  MoveL 2483 to (5.96, 26.09, 110) mm, rotated rx 180 ry 0 rz 180 deg; joints [-156.697, -51.391, -91.658, 28.324, 56.489, -16.571]
  Call Extruder(23411.01401)
  MoveL 2484 to (0, 26.77, 110) mm, rotated rx 180 ry 0 rz 180 deg; joints [-156.245, -51.047, -92.58, 28.662, 57.126, -16.525]
  Call Extruder(23420.37911)
  MoveL 2485 to (-5.96, 26.09, 110) mm, rotated rx 180 ry 0 rz 180 deg; joints [-155.969, -50.675, -93.588, 28.78, 57.762, -16.332]
  Call Extruder(23429.74391)
  MoveL 2486 to (-11.61, 24.12, 110) mm, rotated rx -180 ry 0 rz 180 deg; joints [-155.891, -50.295, -94.633, 28.669, 58.366, -16.002]
  Call Extruder(23439.10883)
  MoveL 2487 to (-16.69, 20.93, 110) mm, rotated rx 180 ry 0 rz -180 deg; joints [-156.025, -49.925, -95.662, 28.327, 58.909, -15.555]
  Call Extruder(23448.47404)
  MoveL 2488 to (-20.93, 16.69, 110) mm, rotated rx 180 ry 0 rz -180 deg; joints [-156.374, -49.585, -96.624, 27.76, 59.366, -15.014]
  Call Extruder(23457.83895)
  MoveL 2489 to (-24.11, 11.61, 110) mm, rotated rx 180 ry 0 rz 180 deg; joints [-156.928, -49.29, -97.469, 26.989, 59.714, -14.405]
  Call Extruder(23467.20375)
  MoveL 2490 to (-26.09, 5.96, 110) mm, rotated rx 180 ry 0 rz 180 deg; joints [-157.665, -49.055, -98.151, 26.047, 59.935, -13.758]
  Call Extruder(23476.56885)
  MoveL 2491 to (-26.77, 0, 110) mm, rotated rx 180 ry 0 rz 180 deg; joints [-158.546, -48.891, -98.632, 24.978, 60.016, -13.105]
  Call Extruder(23481.35759)
  MoveL 2492 to (-26.42, -3.05, 110) mm, rotated rx -180 ry 0 rz 180 deg; joints [-159.044, -48.846, -98.764, 24.396, 59.984, -12.783]
  Set speed (130.0 mm/s)
  MoveL 2493 to (-41.86, -6.3, 110) mm, rotated rx 180 ry 0 rz -180 deg; joints [-158.606, -47.984, -101.368, 24.484, 61.665, -12.196]
  Call Extruder(23486.35544)
  Set speed (60.0 mm/s)
  MoveL 2494 to (-41.5, -9.47, 110) mm, rotated rx 180 ry 0 rz 180 deg; joints [-159.151, -47.941, -101.503, 23.858, 61.634, -11.866]
  Call Extruder(23501.25108)
  MoveL 2495 to (-38.36, -18.47, 110) mm, rotated rx 180 ry 0 rz 180 deg; joints [-160.835, -47.935, -101.523, 21.976, 61.313, -10.963]
  Call Extruder(23516.14694)
  MoveL 2496 to (-33.29, -26.54, 110) mm, rotated rx -180 ry 0 rz 180 deg; joints [-162.466, -48.056, -101.146, 20.195, 60.776, -10.181]
  Call Extruder(23531.04275)
  MoveL 2497 to (-26.54, -33.28, 110) mm, rotated rx -180 ry 0 rz -180 deg; joints [-163.93, -48.301, -100.397, 18.631, 60.049, -9.555]
  Call Extruder(23545.93861)
  MoveL 2498 to (-18.47, -38.36, 110) mm, rotated rx 180 ry 0 rz 180 deg; joints [-165.137, -48.658, -99.32, 17.381, 59.17, -9.114]
  Call Extruder(23560.83426)
  MoveL 2499 to (-9.47, -41.51, 110) mm, rotated rx -180 ry 0 rz 180 deg; joints [-166.024, -49.114, -97.98, 16.512, 58.184, -8.882]
  Call Extruder(23575.73014)
  MoveL 2500 to (0, -42.57, 110) mm, rotated rx 180 ry 0 rz 180 deg; joints [-166.562, -49.645, -96.451, 16.06, 57.144, -8.877]
  Call Extruder(23586.78613)
  MoveL 2501 to (7.03, -41.78, 110) mm, rotated rx -180 ry 0 rz -180 deg; joints [-166.699, -50.076, -95.239, 16.04, 56.372, -9.047]
  Call Extruder(23590.62601)
  MoveL 2502 to (9.47, -41.51, 110) mm, rotated rx 180 ry 0 rz 180 deg; joints [-166.745, -50.229, -94.815, 16.035, 56.104, -9.106]
  Call Extruder(23605.52167)
  MoveL 2503 to (18.47, -38.36, 110) mm, rotated rx -180 ry 0 rz 180 deg; joints [-166.591, -50.834, -93.155, 16.421, 55.117, -9.567]
  Call Extruder(23620.41752)
  MoveL 2504 to (26.54, -33.29, 110) mm, rotated rx -180 ry 0 rz 180 deg; joints [-166.133, -51.431, -91.553, 17.181, 54.233, -10.244]
  Call Extruder(23635.31333)
  MoveL 2505 to (33.28, -26.54, 110) mm, rotated rx -180 ry 0 rz 180 deg; joints [-165.409, -51.988, -90.083, 18.264, 53.497, -11.107]
  Call Extruder(23650.20919)
  MoveL 2506 to (38.36, -18.47, 110) mm, rotated rx 180 ry 0 rz 180 deg; joints [-164.468, -52.477, -88.814, 19.605, 52.948, -12.112]
  Call Extruder(23665.10484)
  MoveL 2507 to (41.51, -9.47, 110) mm, rotated rx 180 ry 0 rz 180 deg; joints [-163.355, -52.87, -87.803, 21.131, 52.614, -13.207]
  Call Extruder(23680.00071)
  MoveL 2508 to (42.57, 0, 110) mm, rotated rx 180 ry 0 rz 180 deg; joints [-162.12, -53.148, -87.097, 22.765, 52.51, -14.327]
  Call Extruder(23694.89659)
  MoveL 2509 to (41.5, 9.47, 110) mm, rotated rx 180 ry 0 rz 180 deg; joints [-160.81, -53.294, -86.726, 24.427, 52.64, -15.409]
  Call Extruder(23709.79225)
  MoveL 2510 to (38.36, 18.47, 110) mm, rotated rx 180 ry 0 rz 180 deg; joints [-159.475, -53.301, -86.709, 26.043, 52.996, -16.389]
  Call Extruder(23724.68809)
  MoveL 2511 to (33.28, 26.54, 110) mm, rotated rx -180 ry 0 rz -180 deg; joints [-158.16, -53.168, -87.044, 27.544, 53.558, -17.213]
  Call Extruder(23739.58392)
  MoveL 2512 to (26.54, 33.28, 110) mm, rotated rx 180 ry 0 rz 180 deg; joints [-156.916, -52.903, -87.719, 28.872, 54.293, -17.839]
  Call Extruder(23754.47976)
  MoveL 2513 to (18.47, 38.36, 110) mm, rotated rx 180 ry 0 rz -180 deg; joints [-155.789, -52.52, -88.701, 29.976, 55.164, -18.236]
  Call Extruder(23769.37542)
  MoveL 2514 to (9.47, 41.51, 110) mm, rotated rx 180 ry 0 rz 180 deg; joints [-154.828, -52.04, -89.947, 30.816, 56.127, -18.39]
  Call Extruder(23784.27129)
  MoveL 2515 to (0, 42.57, 110) mm, rotated rx 180 ry 0 rz 180 deg; joints [-154.081, -51.489, -91.4, 31.359, 57.134, -18.3]
  Call Extruder(23799.16717)
  MoveL 2516 to (-9.47, 41.51, 110) mm, rotated rx 180 ry 0 rz 180 deg; joints [-153.594, -50.894, -92.992, 31.576, 58.137, -17.976]
  Call Extruder(23814.06282)
  MoveL 2517 to (-18.47, 38.36, 110) mm, rotated rx 180 ry 0 rz -180 deg; joints [-153.408, -50.288, -94.65, 31.448, 59.09, -17.44]
  Call Extruder(23828.95867)
  MoveL 2518 to (-26.54, 33.29, 110) mm, rotated rx 180 ry 0 rz 180 deg; joints [-153.557, -49.701, -96.292, 30.961, 59.949, -16.722]
  Call Extruder(23843.85449)
  MoveL 2519 to (-33.28, 26.54, 110) mm, rotated rx 180 ry 0 rz -180 deg; joints [-154.059, -49.163, -97.835, 30.115, 60.674, -15.859]
  Call Extruder(23858.75034)
  MoveL 2520 to (-38.36, 18.47, 110) mm, rotated rx -180 ry 0 rz 180 deg; joints [-154.913, -48.699, -99.198, 28.928, 61.229, -14.896]
  Call Extruder(23873.64600)
  MoveL 2521 to (-41.5, 9.47, 110) mm, rotated rx 180 ry 0 rz 180 deg; joints [-156.091, -48.331, -100.303, 27.439, 61.587, -13.877]
  Call Extruder(23888.54187)
  MoveL 2522 to (-42.57, 0, 110) mm, rotated rx 180 ry 0 rz -180 deg; joints [-157.533, -48.075, -101.088, 25.717, 61.726, -12.852]
  Call Extruder(23896.09615)
  MoveL 2523 to (-42.03, -4.8, 110) mm, rotated rx -180 ry 0 rz 180 deg; joints [-158.35, -48.005, -101.304, 24.777, 61.679, -12.351]
  Set speed (130.0 mm/s)
  MoveL 2524 to (-54.1, -7.67, 110) mm, rotated rx -180 ry 0 rz 180 deg; joints [-158.024, -47.368, -103.323, 24.834, 63.002, -11.865]
  Call Extruder(23900.16878)
  Set speed (30.0 mm/s)
  MoveL 2525 to (-53.59, -12.23, 110) mm, rotated rx 180 ry 0 rz 180 deg; joints [-158.835, -47.307, -103.518, 23.914, 62.961, -11.397]
  Call Extruder(23911.09891)
  MoveL 2526 to (-49.52, -23.85, 110) mm, rotated rx 180 ry 0 rz 180 deg; joints [-161.095, -47.299, -103.544, 21.413, 62.554, -10.246]
  Call Extruder(23922.02920)
  MoveL 2527 to (-42.98, -34.27, 110) mm, rotated rx 180 ry 0 rz 180 deg; joints [-163.275, -47.453, -103.047, 19.047, 61.862, -9.248]
  Call Extruder(23932.95931)
  MoveL 2528 to (-34.27, -42.98, 110) mm, rotated rx -180 ry 0 rz 180 deg; joints [-165.21, -47.763, -102.059, 16.983, 60.92, -8.443]
  Call Extruder(23943.88960)
  MoveL 2529 to (-23.85, -49.52, 110) mm, rotated rx 180 ry 0 rz 180 deg; joints [-166.774, -48.219, -100.647, 15.354, 59.779, -7.869]
  Call Extruder(23954.81973)
  MoveL 2530 to (-12.23, -53.59, 110) mm, rotated rx -180 ry 0 rz 180 deg; joints [-167.889, -48.801, -98.897, 14.245, 58.5, -7.556]
  Call Extruder(23965.74996)
  MoveL 2531 to (0, -54.97, 110) mm, rotated rx 180 ry 0 rz 180 deg; joints [-168.526, -49.485, -96.91, 13.696, 57.152, -7.53]
  Call Extruder(23973.26563)
  MoveL 2532 to (8.41, -54.02, 110) mm, rotated rx -180 ry 0 rz -180 deg; joints [-168.645, -49.998, -95.458, 13.702, 56.225, -7.719]
  Call Extruder(23976.68018)
  MoveL 2533 to (12.23, -53.59, 110) mm, rotated rx -180 ry 0 rz 180 deg; joints [-168.697, -50.237, -94.793, 13.708, 55.804, -7.806]
  Call Extruder(23987.61032)
  MoveL 2534 to (23.85, -49.53, 110) mm, rotated rx 180 ry 0 rz 180 deg; joints [-168.436, -51.019, -92.655, 14.25, 54.524, -8.384]
  Call Extruder(23998.54060)
  MoveL 2535 to (34.27, -42.98, 110) mm, rotated rx 180 ry 0 rz 180 deg; joints [-167.797, -51.793, -90.596, 15.27, 53.379, -9.249]
  Call Extruder(24009.47072)
  MoveL 2536 to (42.98, -34.27, 110) mm, rotated rx 180 ry 0 rz 180 deg; joints [-166.837, -52.516, -88.711, 16.697, 52.427, -10.365]
  Call Extruder(24020.40100)
  MoveL 2537 to (49.53, -23.85, 110) mm, rotated rx -180 ry 0 rz 180 deg; joints [-165.618, -53.151, -87.087, 18.447, 51.717, -11.676]
  Call Extruder(24031.33113)
  MoveL 2538 to (53.59, -12.23, 110) mm, rotated rx -180 ry 0 rz -180 deg; joints [-164.2, -53.663, -85.795, 20.423, 51.285, -13.11]
  Call Extruder(24042.26136)
  MoveL 2539 to (54.97, 0, 110) mm, rotated rx -180 ry 0 rz 180 deg; joints [-162.641, -54.025, -84.892, 22.525, 51.154, -14.581]
  Call Extruder(24053.19158)
  MoveL 2540 to (53.59, 12.23, 110) mm, rotated rx 180 ry 0 rz 180 deg; joints [-160.996, -54.215, -84.418, 24.65, 51.329, -16]
  Call Extruder(24064.12172)
  MoveL 2541 to (49.52, 23.85, 110) mm, rotated rx 180 ry 0 rz -180 deg; joints [-159.322, -54.224, -84.396, 26.703, 51.796, -17.28]
  Call Extruder(24075.05200)
  MoveL 2542 to (42.98, 34.27, 110) mm, rotated rx 180 ry 0 rz 180 deg; joints [-157.673, -54.052, -84.825, 28.599, 52.528, -18.35]
  Call Extruder(24085.98212)
  MoveL 2543 to (34.27, 42.98, 110) mm, rotated rx 180 ry 0 rz 180 deg; joints [-156.102, -53.706, -85.687, 30.269, 53.483, -19.152]
  Call Extruder(24096.91240)
  MoveL 2544 to (23.85, 49.52, 110) mm, rotated rx -180 ry 0 rz 180 deg; joints [-154.667, -53.208, -86.943, 31.658, 54.609, -19.652]
  Call Extruder(24107.84254)
  MoveL 2545 to (12.23, 53.59, 110) mm, rotated rx -180 ry 0 rz 180 deg; joints [-153.426, -52.584, -88.537, 32.722, 55.85, -19.834]
  Call Extruder(24118.77276)
  MoveL 2546 to (0, 54.97, 110) mm, rotated rx 180 ry 0 rz 180 deg; joints [-152.438, -51.868, -90.399, 33.423, 57.144, -19.7]
  Call Extruder(24129.70298)
  MoveL 2547 to (-12.23, 53.59, 110) mm, rotated rx 180 ry 0 rz 180 deg; joints [-151.764, -51.097, -92.445, 33.73, 58.431, -19.267]
  Call Extruder(24140.63312)
  MoveL 2548 to (-23.85, 49.52, 110) mm, rotated rx 180 ry 0 rz 180 deg; joints [-151.463, -50.313, -94.58, 33.612, 59.654, -18.563]
  Call Extruder(24151.56340)
  MoveL 2549 to (-34.27, 42.98, 110) mm, rotated rx 180 ry 0 rz 180 deg; joints [-151.589, -49.557, -96.704, 33.044, 60.756, -17.63]
  Call Extruder(24162.49352)
  MoveL 2550 to (-42.98, 34.27, 110) mm, rotated rx 180 ry 0 rz -180 deg; joints [-152.179, -48.865, -98.708, 32.013, 61.69, -16.514]
  Call Extruder(24173.42380)
  MoveL 2551 to (-49.53, 23.85, 110) mm, rotated rx -180 ry 0 rz -180 deg; joints [-153.248, -48.271, -100.487, 30.523, 62.41, -15.273]
  Call Extruder(24184.35394)
  MoveL 2552 to (-53.59, 12.23, 110) mm, rotated rx -180 ry 0 rz -180 deg; joints [-154.769, -47.802, -101.937, 28.615, 62.879, -13.966]
  Call Extruder(24195.28416)
  MoveL 2553 to (-54.97, 0, 110) mm, rotated rx 180 ry 0 rz -180 deg; joints [-156.673, -47.477, -102.97, 26.369, 63.069, -12.655]
  Call Extruder(24200.80978)
  MoveL 2554 to (-54.27, -6.18, 110) mm, rotated rx 180 ry 0 rz 180 deg; joints [-157.76, -47.388, -103.256, 25.134, 63.015, -12.018]
  Set speed (130.0 mm/s)
  MoveL 2555 to (-49.9, -9.51, 110) mm, rotated rx -180 ry 0 rz 180 deg; joints [-158.616, -47.532, -102.794, 24.26, 62.549, -11.736]
  MoveL 2556 to (2.97, -12.99, 110) mm, rotated rx -180 ry 0 rz -180 deg; joints [-162.152, -50.315, -94.576, 21.484, 56.807, -12.16]
  Call Extruder(24205.47337)
  Set speed (80.0 mm/s)
  MoveL 2557 to (5.78, -12.01, 110) mm, rotated rx -180 ry 0 rz 180 deg; joints [-162.141, -50.504, -94.055, 21.578, 56.501, -12.313]
  Call Extruder(24210.13699)
  MoveL 2558 to (8.31, -10.42, 110) mm, rotated rx -180 ry 0 rz -180 deg; joints [-162.027, -50.69, -93.547, 21.791, 56.227, -12.53]
  Call Extruder(24214.80118)
  MoveL 2559 to (10.42, -8.31, 110) mm, rotated rx 180 ry 0 rz 180 deg; joints [-161.819, -50.862, -93.079, 22.109, 55.998, -12.799]
  Call Extruder(24219.46481)
  MoveL 2560 to (12.01, -5.78, 110) mm, rotated rx -180 ry 0 rz 180 deg; joints [-161.529, -51.013, -92.673, 22.517, 55.826, -13.108]
  Call Extruder(24224.12838)
  MoveL 2561 to (13, -2.97, 110) mm, rotated rx -180 ry 0 rz -180 deg; joints [-161.171, -51.133, -92.348, 22.992, 55.72, -13.441]
  Call Extruder(24228.79233)
  MoveL 2562 to (13.33, 0, 110) mm, rotated rx -180 ry 0 rz 180 deg; joints [-160.763, -51.218, -92.12, 23.51, 55.685, -13.779]
  Call Extruder(24233.45628)
  MoveL 2563 to (12.99, 2.97, 110) mm, rotated rx -180 ry 0 rz 180 deg; joints [-160.324, -51.263, -92, 24.046, 55.722, -14.107]
  Call Extruder(24238.11985)
  MoveL 2564 to (12.01, 5.78, 110) mm, rotated rx 180 ry 0 rz -180 deg; joints [-159.874, -51.265, -91.995, 24.575, 55.83, -14.405]
  Call Extruder(24242.78348)
  MoveL 2565 to (10.42, 8.31, 110) mm, rotated rx 180 ry 0 rz 180 deg; joints [-159.432, -51.225, -92.103, 25.071, 56.002, -14.66]
  Call Extruder(24247.44767)
  MoveL 2566 to (8.31, 10.42, 110) mm, rotated rx 180 ry 0 rz -180 deg; joints [-159.021, -51.144, -92.321, 25.512, 56.23, -14.857]
  Call Extruder(24252.11129)
  MoveL 2567 to (5.78, 12.01, 110) mm, rotated rx 180 ry 0 rz 180 deg; joints [-158.657, -51.026, -92.637, 25.877, 56.502, -14.987]
  Call Extruder(24256.77487)
  MoveL 2568 to (2.97, 13, 110) mm, rotated rx 180 ry 0 rz -180 deg; joints [-158.359, -50.878, -93.036, 26.149, 56.805, -15.045]
  Call Extruder(24261.43882)
  MoveL 2569 to (0, 13.33, 110) mm, rotated rx -180 ry 0 rz -180 deg; joints [-158.143, -50.708, -93.499, 26.314, 57.124, -15.026]
  Call Extruder(24266.10278)
  MoveL 2570 to (-2.97, 13, 110) mm, rotated rx 180 ry 0 rz 180 deg; joints [-158.019, -50.523, -94.003, 26.365, 57.443, -14.934]
  Call Extruder(24270.76634)
  MoveL 2571 to (-5.78, 12.01, 110) mm, rotated rx 180 ry 0 rz 180 deg; joints [-157.997, -50.334, -94.524, 26.296, 57.745, -14.774]
  Call Extruder(24275.42997)
  MoveL 2572 to (-8.31, 10.42, 110) mm, rotated rx -180 ry 0 rz 180 deg; joints [-158.08, -50.149, -95.035, 26.111, 58.018, -14.553]
  Call Extruder(24280.09417)
  MoveL 2573 to (-10.42, 8.31, 110) mm, rotated rx 180 ry 0 rz 180 deg; joints [-158.266, -49.979, -95.511, 25.816, 58.246, -14.284]
  Call Extruder(24284.75779)
  MoveL 2574 to (-12.01, 5.78, 110) mm, rotated rx 180 ry 0 rz 180 deg; joints [-158.549, -49.831, -95.927, 25.423, 58.418, -13.979]
  Call Extruder(24289.42136)
  MoveL 2575 to (-13, 2.97, 110) mm, rotated rx 180 ry 0 rz -180 deg; joints [-158.913, -49.713, -96.261, 24.951, 58.526, -13.654]
  Call Extruder(24294.08531)
  MoveL 2576 to (-13.33, 0, 110) mm, rotated rx 180 ry 0 rz 180 deg; joints [-159.341, -49.63, -96.496, 24.424, 58.565, -13.324]
  Call Extruder(24298.74927)
  MoveL 2577 to (-12.99, -2.97, 110) mm, rotated rx -180 ry 0 rz 180 deg; joints [-159.811, -49.586, -96.62, 23.868, 58.531, -13.006]
  Call Extruder(24303.41283)
  MoveL 2578 to (-12.01, -5.78, 110) mm, rotated rx 180 ry 0 rz 180 deg; joints [-160.294, -49.584, -96.626, 23.314, 58.427, -12.715]
  Call Extruder(24308.07647)
  MoveL 2579 to (-10.42, -8.31, 110) mm, rotated rx 180 ry 0 rz 180 deg; joints [-160.766, -49.623, -96.514, 22.791, 58.257, -12.465]
  Call Extruder(24312.74065)
  MoveL 2580 to (-8.31, -10.42, 110) mm, rotated rx 180 ry 0 rz 180 deg; joints [-161.2, -49.703, -96.289, 22.327, 58.03, -12.268]
  Call Extruder(24317.40429)
  MoveL 2581 to (-5.78, -12.01, 110) mm, rotated rx 180 ry 0 rz 180 deg; joints [-161.572, -49.818, -95.964, 21.947, 57.757, -12.133]
  Call Extruder(24322.06785)
  MoveL 2582 to (-2.97, -13, 110) mm, rotated rx 180 ry 0 rz 180 deg; joints [-161.863, -49.963, -95.555, 21.673, 57.452, -12.068]
  Call Extruder(24326.73181)
  MoveL 2583 to (0, -13.33, 110) mm, rotated rx 180 ry 0 rz -180 deg; joints [-162.059, -50.132, -95.084, 21.516, 57.13, -12.077]
  Call Extruder(24331.39575)
  MoveL 2584 to (2.97, -12.99, 110) mm, rotated rx -180 ry 0 rz -180 deg; joints [-162.152, -50.315, -94.576, 21.484, 56.807, -12.16]
  Set speed (130.0 mm/s)
  MoveL 2585 to (2.97, -12.99, 115) mm, rotated rx 180 ry 0 rz -180 deg; joints [-162.152, -49.558, -94.868, 21.597, 56.374, -12.365]
  MoveL 2586 to (-26.25, -4.54, 115) mm, rotated rx 180 ry 0 rz 180 deg; joints [-159.288, -48.032, -99.127, 24.229, 59.519, -12.859]
  Call Extruder(24333.62836)
  Set speed (60.0 mm/s)
  MoveL 2587 to (-26.09, -5.96, 115) mm, rotated rx 180 ry 0 rz 180 deg; joints [-159.522, -48.012, -99.186, 23.955, 59.502, -12.707]
  Call Extruder(24342.99315)
  MoveL 2588 to (-24.11, -11.61, 115) mm, rotated rx 180 ry 0 rz 180 deg; joints [-160.532, -48.007, -99.199, 22.808, 59.293, -12.12]
  Call Extruder(24352.35808)
  MoveL 2589 to (-20.93, -16.69, 115) mm, rotated rx -180 ry 0 rz 180 deg; joints [-161.513, -48.087, -98.968, 21.723, 58.951, -11.612]
  Call Extruder(24361.72328)
  MoveL 2590 to (-16.69, -20.93, 115) mm, rotated rx 180 ry 0 rz 180 deg; joints [-162.406, -48.248, -98.507, 20.764, 58.495, -11.207]
  Call Extruder(24371.08820)
  MoveL 2591 to (-11.61, -24.12, 115) mm, rotated rx 180 ry 0 rz 180 deg; joints [-163.159, -48.482, -97.842, 19.988, 57.946, -10.926]
  Call Extruder(24380.45299)
  MoveL 2592 to (-5.96, -26.09, 115) mm, rotated rx -180 ry 0 rz 180 deg; joints [-163.733, -48.779, -97.01, 19.435, 57.334, -10.783]
  Call Extruder(24389.81809)
  MoveL 2593 to (0, -26.77, 115) mm, rotated rx 180 ry 0 rz 180 deg; joints [-164.103, -49.123, -96.056, 19.133, 56.689, -10.787]
  Call Extruder(24399.18321)
  MoveL 2594 to (5.96, -26.09, 115) mm, rotated rx -180 ry 0 rz 180 deg; joints [-164.258, -49.498, -95.029, 19.092, 56.044, -10.942]
  Call Extruder(24408.54800)
  MoveL 2595 to (11.61, -24.11, 115) mm, rotated rx -180 ry 0 rz 180 deg; joints [-164.201, -49.886, -93.982, 19.307, 55.433, -11.242]
  Call Extruder(24417.91291)
  MoveL 2596 to (16.69, -20.93, 115) mm, rotated rx 180 ry 0 rz 180 deg; joints [-163.944, -50.267, -92.967, 19.762, 54.886, -11.676]
  Call Extruder(24427.27812)
  MoveL 2597 to (20.93, -16.69, 115) mm, rotated rx 180 ry 0 rz 180 deg; joints [-163.508, -50.622, -92.033, 20.426, 54.433, -12.222]
  Call Extruder(24436.64304)
  MoveL 2598 to (24.12, -11.61, 115) mm, rotated rx 180 ry 0 rz 180 deg; joints [-162.92, -50.932, -91.224, 21.261, 54.094, -12.854]
  Call Extruder(24446.00784)
  MoveL 2599 to (26.09, -5.96, 115) mm, rotated rx -180 ry 0 rz -180 deg; joints [-162.209, -51.181, -90.579, 22.222, 53.889, -13.538]
  Call Extruder(24455.37293)
  MoveL 2600 to (26.77, 0, 115) mm, rotated rx -180 ry 0 rz -180 deg; joints [-161.41, -51.356, -90.128, 23.261, 53.826, -14.237]
  Call Extruder(24464.73804)
  MoveL 2601 to (26.09, 5.96, 115) mm, rotated rx -180 ry 0 rz -180 deg; joints [-160.556, -51.449, -89.891, 24.327, 53.909, -14.912]
  Call Extruder(24474.10285)
  MoveL 2602 to (24.11, 11.61, 115) mm, rotated rx -180 ry 0 rz 180 deg; joints [-159.683, -51.453, -89.88, 25.37, 54.132, -15.528]
  Call Extruder(24483.46775)
  MoveL 2603 to (20.93, 16.69, 115) mm, rotated rx 180 ry 0 rz 180 deg; joints [-158.826, -51.369, -90.095, 26.345, 54.483, -16.05]
  Call Extruder(24492.83297)
  MoveL 2604 to (16.69, 20.93, 115) mm, rotated rx 180 ry 0 rz 180 deg; joints [-158.019, -51.202, -90.525, 27.209, 54.944, -16.452]
  Call Extruder(24502.19787)
  MoveL 2605 to (11.61, 24.12, 115) mm, rotated rx -180 ry 0 rz 180 deg; joints [-157.299, -50.96, -91.152, 27.926, 55.49, -16.715]
  Call Extruder(24511.56268)
  MoveL 2606 to (5.96, 26.09, 115) mm, rotated rx -180 ry 0 rz 180 deg; joints [-156.697, -50.655, -91.946, 28.466, 56.095, -16.827]
  Call Extruder(24520.92778)
  MoveL 2607 to (0, 26.77, 115) mm, rotated rx 180 ry 0 rz -180 deg; joints [-156.245, -50.304, -92.87, 28.804, 56.728, -16.786]
  Call Extruder(24530.29289)
  MoveL 2608 to (-5.96, 26.09, 115) mm, rotated rx 180 ry 0 rz 180 deg; joints [-155.969, -49.925, -93.879, 28.921, 57.359, -16.594]
  Call Extruder(24539.65768)
  MoveL 2609 to (-11.61, 24.12, 115) mm, rotated rx 180 ry 0 rz -180 deg; joints [-155.891, -49.537, -94.925, 28.809, 57.958, -16.266]
  Call Extruder(24549.02260)
  MoveL 2610 to (-16.69, 20.93, 115) mm, rotated rx 180 ry 0 rz -180 deg; joints [-156.025, -49.159, -95.956, 28.463, 58.494, -15.818]
  Call Extruder(24558.38781)
  MoveL 2611 to (-20.93, 16.69, 115) mm, rotated rx 180 ry 0 rz 180 deg; joints [-156.374, -48.811, -96.92, 27.894, 58.944, -15.273]
  Call Extruder(24567.75272)
  MoveL 2612 to (-24.11, 11.61, 115) mm, rotated rx -180 ry 0 rz 180 deg; joints [-156.928, -48.509, -97.766, 27.119, 59.283, -14.66]
  Call Extruder(24577.11752)
  MoveL 2613 to (-26.09, 5.96, 115) mm, rotated rx 180 ry 0 rz -180 deg; joints [-157.665, -48.268, -98.449, 26.172, 59.496, -14.007]
  Call Extruder(24586.48263)
  MoveL 2614 to (-26.77, 0, 115) mm, rotated rx 180 ry 0 rz -180 deg; joints [-158.546, -48.1, -98.932, 25.099, 59.571, -13.346]
  Call Extruder(24591.27137)
  MoveL 2615 to (-26.42, -3.05, 115) mm, rotated rx 180 ry 0 rz 180 deg; joints [-159.044, -48.054, -99.064, 24.515, 59.536, -13.019]
  Set speed (130.0 mm/s)
  MoveL 2616 to (-41.86, -6.3, 115) mm, rotated rx -180 ry 0 rz 180 deg; joints [-158.606, -47.168, -101.674, 24.6, 61.201, -12.438]
  Call Extruder(24596.26921)
  Set speed (60.0 mm/s)
  MoveL 2617 to (-41.51, -9.47, 115) mm, rotated rx 180 ry 0 rz -180 deg; joints [-159.151, -47.124, -101.809, 23.97, 61.167, -12.102]
  Call Extruder(24611.16485)
  MoveL 2618 to (-38.36, -18.47, 115) mm, rotated rx 180 ry 0 rz 180 deg; joints [-160.835, -47.117, -101.829, 22.082, 60.839, -11.182]
  Call Extruder(24626.06071)
  MoveL 2619 to (-33.28, -26.54, 115) mm, rotated rx 180 ry 0 rz 180 deg; joints [-162.466, -47.242, -101.451, 20.294, 60.299, -10.383]
  Call Extruder(24640.95653)
  MoveL 2620 to (-26.54, -33.28, 115) mm, rotated rx -180 ry 0 rz -180 deg; joints [-163.93, -47.494, -100.7, 18.725, 59.572, -9.741]
  Call Extruder(24655.85238)
  MoveL 2621 to (-18.47, -38.36, 115) mm, rotated rx -180 ry 0 rz 180 deg; joints [-165.137, -47.862, -99.621, 17.471, 58.697, -9.287]
  Call Extruder(24670.74803)
  MoveL 2622 to (-9.47, -41.5, 115) mm, rotated rx 180 ry 0 rz 180 deg; joints [-166.024, -48.328, -98.278, 16.599, 57.718, -9.046]
  Call Extruder(24685.64390)
  MoveL 2623 to (0, -42.57, 115) mm, rotated rx 180 ry 0 rz 180 deg; joints [-166.562, -48.873, -96.746, 16.146, 56.686, -9.035]
  Call Extruder(24697.35594)
  MoveL 2624 to (7.45, -41.73, 115) mm, rotated rx 180 ry 0 rz 180 deg; joints [-166.707, -49.34, -95.46, 16.126, 55.876, -9.213]
  Call Extruder(24700.53978)
  MoveL 2625 to (9.47, -41.51, 115) mm, rotated rx 180 ry 0 rz 180 deg; joints [-166.745, -49.469, -95.108, 16.123, 55.656, -9.262]
  Call Extruder(24715.43544)
  MoveL 2626 to (18.47, -38.36, 115) mm, rotated rx -180 ry 0 rz 180 deg; joints [-166.591, -50.087, -93.445, 16.512, 54.678, -9.725]
  Call Extruder(24730.33128)
  MoveL 2627 to (26.54, -33.28, 115) mm, rotated rx 180 ry 0 rz 180 deg; joints [-166.133, -50.695, -91.84, 17.277, 53.805, -10.408]
  Call Extruder(24745.22710)
  MoveL 2628 to (33.29, -26.54, 115) mm, rotated rx 180 ry 0 rz -180 deg; joints [-165.409, -51.263, -90.369, 18.367, 53.08, -11.279]
  Call Extruder(24760.12296)
  MoveL 2629 to (38.36, -18.47, 115) mm, rotated rx 180 ry 0 rz 180 deg; joints [-164.468, -51.759, -89.098, 19.715, 52.541, -12.295]
  Call Extruder(24775.01861)
  MoveL 2630 to (41.5, -9.47, 115) mm, rotated rx -180 ry 0 rz 180 deg; joints [-163.355, -52.159, -88.087, 21.25, 52.215, -13.402]
  Call Extruder(24789.91448)
  MoveL 2631 to (42.57, 0, 115) mm, rotated rx 180 ry 0 rz 180 deg; joints [-162.12, -52.441, -87.38, 22.892, 52.119, -14.535]
  Call Extruder(24804.81036)
  MoveL 2632 to (41.51, 9.47, 115) mm, rotated rx 180 ry 0 rz 180 deg; joints [-160.81, -52.589, -87.009, 24.562, 52.256, -15.629]
  Call Extruder(24819.70602)
  MoveL 2633 to (38.36, 18.47, 115) mm, rotated rx 180 ry 0 rz 180 deg; joints [-159.475, -52.596, -86.991, 26.184, 52.618, -16.622]
  Call Extruder(24834.60186)
  MoveL 2634 to (33.29, 26.54, 115) mm, rotated rx -180 ry 0 rz -180 deg; joints [-158.16, -52.462, -87.328, 27.69, 53.183, -17.458]
  Call Extruder(24849.49768)
  MoveL 2635 to (26.54, 33.28, 115) mm, rotated rx 180 ry 0 rz 180 deg; joints [-156.916, -52.193, -88.002, 29.021, 53.92, -18.094]
  Call Extruder(24864.39353)
  MoveL 2636 to (18.47, 38.36, 115) mm, rotated rx 180 ry 0 rz -180 deg; joints [-155.789, -51.804, -88.985, 30.128, 54.79, -18.5]
  Call Extruder(24879.28919)
  MoveL 2637 to (9.47, 41.5, 115) mm, rotated rx 180 ry 0 rz 180 deg; joints [-154.828, -51.316, -90.233, 30.968, 55.75, -18.662]
  Call Extruder(24894.18507)
  MoveL 2638 to (0, 42.57, 115) mm, rotated rx 180 ry 0 rz 180 deg; joints [-154.081, -50.754, -91.687, 31.51, 56.752, -18.578]
  Call Extruder(24909.08094)
  MoveL 2639 to (-9.47, 41.51, 115) mm, rotated rx 180 ry 0 rz 180 deg; joints [-153.594, -50.148, -93.282, 31.726, 57.749, -18.258]
  Call Extruder(24923.97659)
  MoveL 2640 to (-18.47, 38.36, 115) mm, rotated rx -180 ry 0 rz -180 deg; joints [-153.408, -49.53, -94.943, 31.595, 58.693, -17.725]
  Call Extruder(24938.87244)
  MoveL 2641 to (-26.54, 33.29, 115) mm, rotated rx 180 ry 0 rz 180 deg; joints [-153.557, -48.93, -96.587, 31.104, 59.541, -17.006]
  Call Extruder(24953.76826)
  MoveL 2642 to (-33.28, 26.54, 115) mm, rotated rx 180 ry 0 rz 180 deg; joints [-154.059, -48.379, -98.133, 30.254, 60.254, -16.14]
  Call Extruder(24968.66411)
  MoveL 2643 to (-38.36, 18.47, 115) mm, rotated rx -180 ry 0 rz -180 deg; joints [-154.913, -47.904, -99.499, 29.061, 60.796, -15.17]
  Call Extruder(24983.55977)
  MoveL 2644 to (-41.5, 9.47, 115) mm, rotated rx 180 ry 0 rz -180 deg; joints [-156.091, -47.526, -100.607, 27.565, 61.141, -14.142]
  Call Extruder(24998.45564)
  MoveL 2645 to (-42.57, 0, 115) mm, rotated rx 180 ry 0 rz -180 deg; joints [-157.533, -47.262, -101.393, 25.837, 61.268, -13.103]
  Call Extruder(25006.00993)
  MoveL 2646 to (-42.03, -4.8, 115) mm, rotated rx -180 ry 0 rz 180 deg; joints [-158.35, -47.19, -101.609, 24.894, 61.217, -12.595]
  Set speed (130.0 mm/s)
  MoveL 2647 to (-54.1, -7.67, 115) mm, rotated rx 180 ry 0 rz -180 deg; joints [-158.024, -46.533, -103.633, 24.948, 62.526, -12.113]
  Call Extruder(25010.08255)
  Set speed (30.0 mm/s)
  MoveL 2648 to (-53.59, -12.23, 115) mm, rotated rx 180 ry 0 rz -180 deg; joints [-158.835, -46.47, -103.829, 24.024, 62.481, -11.637]
  Call Extruder(25021.01269)
  MoveL 2649 to (-49.53, -23.85, 115) mm, rotated rx -180 ry 0 rz 180 deg; joints [-161.095, -46.462, -103.855, 21.514, 62.064, -10.463]
  Call Extruder(25031.94297)
  MoveL 2650 to (-42.98, -34.27, 115) mm, rotated rx 180 ry 0 rz 180 deg; joints [-163.275, -46.621, -103.356, 19.14, 61.368, -9.442]
  Call Extruder(25042.87309)
  MoveL 2651 to (-34.27, -42.98, 115) mm, rotated rx -180 ry 0 rz 180 deg; joints [-165.21, -46.941, -102.367, 17.068, 60.428, -8.616]
  Call Extruder(25053.80337)
  MoveL 2652 to (-23.85, -49.53, 115) mm, rotated rx -180 ry 0 rz 180 deg; joints [-166.774, -47.41, -100.951, 15.433, 59.292, -8.024]
  Call Extruder(25064.73351)
  MoveL 2653 to (-12.23, -53.59, 115) mm, rotated rx 180 ry 0 rz 180 deg; joints [-167.889, -48.008, -99.197, 14.32, 58.023, -7.699]
  Call Extruder(25075.66373)
  MoveL 2654 to (0, -54.97, 115) mm, rotated rx -180 ry 0 rz 180 deg; joints [-168.526, -48.708, -97.206, 13.77, 56.686, -7.666]
  Call Extruder(25083.55224)
  MoveL 2655 to (8.83, -53.97, 115) mm, rotated rx -180 ry 0 rz -180 deg; joints [-168.651, -49.26, -95.679, 13.778, 55.722, -7.863]
  Call Extruder(25086.59395)
  MoveL 2656 to (12.23, -53.59, 115) mm, rotated rx -180 ry 0 rz 180 deg; joints [-168.697, -49.477, -95.086, 13.784, 55.35, -7.94]
  Call Extruder(25097.52409)
  MoveL 2657 to (23.85, -49.53, 115) mm, rotated rx -180 ry 0 rz 180 deg; joints [-168.436, -50.276, -92.944, 14.33, 54.084, -8.522]
  Call Extruder(25108.45437)
  MoveL 2658 to (34.27, -42.98, 115) mm, rotated rx -180 ry 0 rz 180 deg; joints [-167.797, -51.064, -90.882, 15.357, 52.953, -9.395]
  Call Extruder(25119.38449)
  MoveL 2659 to (42.98, -34.27, 115) mm, rotated rx -180 ry 0 rz 180 deg; joints [-166.837, -51.8, -88.996, 16.794, 52.013, -10.523]
  Call Extruder(25130.31477)
  MoveL 2660 to (49.53, -23.85, 115) mm, rotated rx -180 ry 0 rz 180 deg; joints [-165.618, -52.445, -87.37, 18.554, 51.315, -11.848]
  Call Extruder(25141.24491)
  MoveL 2661 to (53.59, -12.23, 115) mm, rotated rx 180 ry 0 rz -180 deg; joints [-164.2, -52.964, -86.077, 20.541, 50.894, -13.298]
  Call Extruder(25152.17513)
  MoveL 2662 to (54.97, 0, 115) mm, rotated rx 180 ry 0 rz 180 deg; joints [-162.641, -53.331, -85.173, 22.654, 50.773, -14.785]
  Call Extruder(25163.10535)
  MoveL 2663 to (53.59, 12.23, 115) mm, rotated rx 180 ry 0 rz 180 deg; joints [-160.996, -53.524, -84.7, 24.788, 50.956, -16.22]
  Call Extruder(25174.03549)
  MoveL 2664 to (49.52, 23.85, 115) mm, rotated rx -180 ry 0 rz -180 deg; joints [-159.322, -53.533, -84.677, 26.849, 51.43, -17.516]
  Call Extruder(25184.96577)
  MoveL 2665 to (42.98, 34.27, 115) mm, rotated rx 180 ry 0 rz 180 deg; joints [-157.673, -53.358, -85.107, 28.751, 52.166, -18.599]
  Call Extruder(25195.89589)
  MoveL 2666 to (34.27, 42.98, 115) mm, rotated rx -180 ry 0 rz -180 deg; joints [-156.102, -53.008, -85.969, 30.426, 53.123, -19.415]
  Call Extruder(25206.82617)
  MoveL 2667 to (23.85, 49.53, 115) mm, rotated rx 180 ry 0 rz -180 deg; joints [-154.667, -52.502, -87.226, 31.818, 54.25, -19.926]
  Call Extruder(25217.75631)
  MoveL 2668 to (12.23, 53.59, 115) mm, rotated rx -180 ry 0 rz 180 deg; joints [-153.426, -51.868, -88.822, 32.882, 55.487, -20.117]
  Call Extruder(25228.68653)
  MoveL 2669 to (0, 54.97, 115) mm, rotated rx 180 ry 0 rz 180 deg; joints [-152.438, -51.14, -90.686, 33.582, 56.776, -19.99]
  Call Extruder(25239.61676)
  MoveL 2670 to (-12.23, 53.59, 115) mm, rotated rx -180 ry 0 rz 180 deg; joints [-151.764, -50.355, -92.734, 33.886, 58.055, -19.563]
  Call Extruder(25250.54689)
  MoveL 2671 to (-23.85, 49.52, 115) mm, rotated rx -180 ry 0 rz 180 deg; joints [-151.463, -49.556, -94.873, 33.764, 59.266, -18.863]
  Call Extruder(25261.47717)
  MoveL 2672 to (-34.27, 42.98, 115) mm, rotated rx 180 ry 0 rz 180 deg; joints [-151.589, -48.782, -96.999, 33.192, 60.356, -17.93]
  Call Extruder(25272.40729)
  MoveL 2673 to (-42.98, 34.27, 115) mm, rotated rx -180 ry 0 rz -180 deg; joints [-152.179, -48.073, -99.008, 32.155, 61.273, -16.812]
  Call Extruder(25283.33757)
  MoveL 2674 to (-49.52, 23.85, 115) mm, rotated rx 180 ry 0 rz 180 deg; joints [-153.248, -47.464, -100.79, 30.659, 61.976, -15.563]
  Call Extruder(25294.26771)
  MoveL 2675 to (-53.59, 12.23, 115) mm, rotated rx 180 ry 0 rz 180 deg; joints [-154.769, -46.981, -102.244, 28.743, 62.428, -14.244]
  Call Extruder(25305.19794)
  MoveL 2676 to (-54.97, 0, 115) mm, rotated rx 180 ry 0 rz -180 deg; joints [-156.673, -46.645, -103.279, 26.488, 62.602, -12.916]
  Call Extruder(25310.72355)
  MoveL 2677 to (-54.27, -6.18, 115) mm, rotated rx 180 ry 0 rz -180 deg; joints [-157.76, -46.554, -103.567, 25.248, 62.541, -12.269]
  Set speed (130.0 mm/s)
  MoveL 2678 to (-49.9, -9.51, 115) mm, rotated rx 180 ry 0 rz 180 deg; joints [-158.616, -46.702, -103.103, 24.372, 62.075, -11.978]
  MoveL 2679 to (2.97, -12.99, 115) mm, rotated rx 180 ry 0 rz -180 deg; joints [-162.152, -49.558, -94.868, 21.597, 56.374, -12.365]
  Call Extruder(25315.38712)
  Set speed (80.0 mm/s)
  MoveL 2680 to (5.78, -12.01, 115) mm, rotated rx 180 ry 0 rz 180 deg; joints [-162.141, -49.751, -94.346, 21.692, 56.071, -12.518]
  Call Extruder(25320.05074)
  MoveL 2681 to (8.31, -10.42, 115) mm, rotated rx -180 ry 0 rz -180 deg; joints [-162.027, -49.94, -93.838, 21.906, 55.8, -12.736]
  Call Extruder(25324.71493)
  MoveL 2682 to (10.42, -8.31, 115) mm, rotated rx 180 ry 0 rz 180 deg; joints [-161.819, -50.116, -93.369, 22.226, 55.575, -13.008]
  Call Extruder(25329.37856)
  MoveL 2683 to (12.01, -5.78, 115) mm, rotated rx 180 ry 0 rz 180 deg; joints [-161.529, -50.269, -92.962, 22.636, 55.407, -13.32]
  Call Extruder(25334.04213)
  MoveL 2684 to (13, -2.97, 115) mm, rotated rx 180 ry 0 rz -180 deg; joints [-161.171, -50.392, -92.637, 23.113, 55.304, -13.656]
  Call Extruder(25338.70608)
  MoveL 2685 to (13.33, 0, 115) mm, rotated rx 180 ry 0 rz 180 deg; joints [-160.763, -50.479, -92.409, 23.634, 55.271, -13.998]
  Call Extruder(25343.37004)
  MoveL 2686 to (13, 2.97, 115) mm, rotated rx 180 ry 0 rz 180 deg; joints [-160.324, -50.524, -92.289, 24.173, 55.311, -14.33]
  Call Extruder(25348.03361)
  MoveL 2687 to (12.01, 5.78, 115) mm, rotated rx -180 ry 0 rz -180 deg; joints [-159.874, -50.527, -92.283, 24.704, 55.42, -14.633]
  Call Extruder(25352.69723)
  MoveL 2688 to (10.42, 8.31, 115) mm, rotated rx 180 ry 0 rz 180 deg; joints [-159.432, -50.485, -92.392, 25.202, 55.594, -14.891]
  Call Extruder(25357.36142)
  MoveL 2689 to (8.31, 10.42, 115) mm, rotated rx -180 ry 0 rz -180 deg; joints [-159.021, -50.403, -92.609, 25.644, 55.822, -15.092]
  Call Extruder(25362.02505)
  MoveL 2690 to (5.78, 12.01, 115) mm, rotated rx 180 ry 0 rz 180 deg; joints [-158.657, -50.283, -92.926, 26.009, 56.094, -15.226]
  Call Extruder(25366.68862)
  MoveL 2691 to (2.97, 13, 115) mm, rotated rx 180 ry 0 rz 180 deg; joints [-158.359, -50.132, -93.326, 26.281, 56.396, -15.286]
  Call Extruder(25371.35258)
  MoveL 2692 to (0, 13.33, 115) mm, rotated rx 180 ry 0 rz 180 deg; joints [-158.143, -49.958, -93.789, 26.447, 56.713, -15.27]
  Call Extruder(25376.01653)
  MoveL 2693 to (-2.97, 12.99, 115) mm, rotated rx 180 ry 0 rz 180 deg; joints [-158.019, -49.77, -94.295, 26.497, 57.029, -15.179]
  Call Extruder(25380.68010)
  MoveL 2694 to (-5.78, 12.01, 115) mm, rotated rx 180 ry 0 rz 180 deg; joints [-157.997, -49.577, -94.816, 26.428, 57.329, -15.018]
  Call Extruder(25385.34373)
  MoveL 2695 to (-8.31, 10.42, 115) mm, rotated rx -180 ry 0 rz 180 deg; joints [-158.08, -49.388, -95.328, 26.241, 57.597, -14.797]
  Call Extruder(25390.00792)
  MoveL 2696 to (-10.42, 8.31, 115) mm, rotated rx 180 ry 0 rz 180 deg; joints [-158.266, -49.214, -95.805, 25.944, 57.822, -14.526]
  Call Extruder(25394.67154)
  MoveL 2697 to (-12.01, 5.78, 115) mm, rotated rx -180 ry 0 rz 180 deg; joints [-158.549, -49.063, -96.221, 25.549, 57.99, -14.219]
  Call Extruder(25399.33511)
  MoveL 2698 to (-12.99, 2.97, 115) mm, rotated rx 180 ry 0 rz -180 deg; joints [-158.913, -48.942, -96.556, 25.075, 58.095, -13.89]
  Call Extruder(25403.99907)
  MoveL 2699 to (-13.33, 0, 115) mm, rotated rx -180 ry 0 rz 180 deg; joints [-159.341, -48.857, -96.792, 24.546, 58.131, -13.557]
  Call Extruder(25408.66302)
  MoveL 2700 to (-12.99, -2.97, 115) mm, rotated rx 180 ry 0 rz 180 deg; joints [-159.811, -48.812, -96.916, 23.988, 58.094, -13.234]
  Call Extruder(25413.32659)
  MoveL 2701 to (-12.01, -5.78, 115) mm, rotated rx 180 ry 0 rz 180 deg; joints [-160.294, -48.81, -96.922, 23.432, 57.988, -12.939]
  Call Extruder(25417.99022)
  MoveL 2702 to (-10.42, -8.31, 115) mm, rotated rx 180 ry 0 rz 180 deg; joints [-160.766, -48.851, -96.809, 22.906, 57.817, -12.683]
  Call Extruder(25422.65441)
  MoveL 2703 to (-8.31, -10.42, 115) mm, rotated rx -180 ry 0 rz 180 deg; joints [-161.2, -48.932, -96.584, 22.441, 57.59, -12.482]
  Call Extruder(25427.31804)
  MoveL 2704 to (-5.78, -12.01, 115) mm, rotated rx 180 ry 0 rz 180 deg; joints [-161.572, -49.049, -96.258, 22.06, 57.317, -12.343]
  Call Extruder(25431.98160)
  MoveL 2705 to (-2.97, -12.99, 115) mm, rotated rx 180 ry 0 rz 180 deg; joints [-161.863, -49.198, -95.849, 21.785, 57.014, -12.276]
  Call Extruder(25436.64555)
  MoveL 2706 to (0, -13.33, 115) mm, rotated rx 180 ry 0 rz -180 deg; joints [-162.059, -49.37, -95.377, 21.628, 56.694, -12.283]
  Call Extruder(25441.30952)
  MoveL 2707 to (2.97, -12.99, 115) mm, rotated rx 180 ry 0 rz -180 deg; joints [-162.152, -49.558, -94.868, 21.597, 56.374, -12.365]
  Set speed (130.0 mm/s)
  MoveL 2708 to (2.97, -12.99, 120) mm, rotated rx 180 ry 0 rz -180 deg; joints [-162.152, -48.802, -95.151, 21.714, 55.934, -12.575]
  MoveL 2709 to (-26.25, -4.54, 120) mm, rotated rx -180 ry 0 rz 180 deg; joints [-159.288, -47.241, -99.418, 24.351, 59.062, -13.099]
  Call Extruder(25443.54214)
  Set speed (60.0 mm/s)
  MoveL 2710 to (-26.09, -5.96, 120) mm, rotated rx 180 ry 0 rz 180 deg; joints [-159.522, -47.22, -99.477, 24.077, 59.044, -12.944]
  Call Extruder(25452.90693)
  MoveL 2711 to (-24.11, -11.61, 120) mm, rotated rx 180 ry 0 rz 180 deg; joints [-160.532, -47.215, -99.489, 22.925, 58.83, -12.347]
  Call Extruder(25462.27185)
  MoveL 2712 to (-20.93, -16.69, 120) mm, rotated rx 180 ry 0 rz 180 deg; joints [-161.513, -47.297, -99.258, 21.835, 58.487, -11.829]
  Call Extruder(25471.63706)
  MoveL 2713 to (-16.69, -20.93, 120) mm, rotated rx 180 ry 0 rz 180 deg; joints [-162.406, -47.462, -98.796, 20.874, 58.03, -11.415]
  Call Extruder(25481.00198)
  MoveL 2714 to (-11.61, -24.12, 120) mm, rotated rx -180 ry 0 rz 180 deg; joints [-163.159, -47.702, -98.13, 20.094, 57.484, -11.125]
  Call Extruder(25490.36677)
  MoveL 2715 to (-5.96, -26.09, 120) mm, rotated rx 180 ry 0 rz 180 deg; joints [-163.733, -48.005, -97.296, 19.54, 56.875, -10.976]
  Call Extruder(25499.73187)
  MoveL 2716 to (0, -26.77, 120) mm, rotated rx 180 ry 0 rz 180 deg; joints [-164.103, -48.357, -96.34, 19.237, 56.235, -10.976]
  Call Extruder(25509.09698)
  MoveL 2717 to (5.96, -26.09, 120) mm, rotated rx 180 ry 0 rz 180 deg; joints [-164.258, -48.741, -95.312, 19.198, 55.596, -11.13]
  Call Extruder(25518.46178)
  MoveL 2718 to (11.61, -24.11, 120) mm, rotated rx 180 ry 0 rz -180 deg; joints [-164.201, -49.137, -94.263, 19.415, 54.992, -11.431]
  Call Extruder(25527.82669)
  MoveL 2719 to (16.69, -20.93, 120) mm, rotated rx 180 ry 0 rz 180 deg; joints [-163.944, -49.526, -93.247, 19.873, 54.452, -11.868]
  Call Extruder(25537.19190)
  MoveL 2720 to (20.93, -16.69, 120) mm, rotated rx -180 ry 0 rz 180 deg; joints [-163.508, -49.887, -92.311, 20.541, 54.005, -12.419]
  Call Extruder(25546.55682)
  MoveL 2721 to (24.12, -11.61, 120) mm, rotated rx 180 ry 0 rz 180 deg; joints [-162.92, -50.202, -91.502, 21.381, 53.673, -13.058]
  Call Extruder(25555.92161)
  MoveL 2722 to (26.09, -5.96, 120) mm, rotated rx -180 ry 0 rz -180 deg; joints [-162.209, -50.456, -90.856, 22.347, 53.474, -13.749]
  Call Extruder(25565.28671)
  MoveL 2723 to (26.77, 0, 120) mm, rotated rx -180 ry 0 rz -180 deg; joints [-161.41, -50.634, -90.404, 23.391, 53.417, -14.456]
  Call Extruder(25574.65182)
  MoveL 2724 to (26.09, 5.96, 120) mm, rotated rx 180 ry 0 rz 180 deg; joints [-160.556, -50.728, -90.167, 24.462, 53.504, -15.14]
  Call Extruder(25584.01662)
  MoveL 2725 to (24.12, 11.61, 120) mm, rotated rx -180 ry 0 rz 180 deg; joints [-159.683, -50.733, -90.156, 25.509, 53.731, -15.764]
  Call Extruder(25593.38153)
  MoveL 2726 to (20.93, 16.69, 120) mm, rotated rx -180 ry 0 rz 180 deg; joints [-158.826, -50.647, -90.371, 26.488, 54.084, -16.294]
  Call Extruder(25602.74674)
  MoveL 2727 to (16.69, 20.93, 120) mm, rotated rx 180 ry 0 rz 180 deg; joints [-158.019, -50.477, -90.802, 27.354, 54.546, -16.704]
  Call Extruder(25612.11165)
  MoveL 2728 to (11.61, 24.11, 120) mm, rotated rx -180 ry 0 rz -180 deg; joints [-157.299, -50.231, -91.43, 28.073, 55.092, -16.973]
  Call Extruder(25621.47646)
  MoveL 2729 to (5.96, 26.09, 120) mm, rotated rx 180 ry 0 rz 180 deg; joints [-156.697, -49.921, -92.225, 28.613, 55.695, -17.09]
  Call Extruder(25630.84156)
  MoveL 2730 to (0, 26.77, 120) mm, rotated rx 180 ry 0 rz 180 deg; joints [-156.245, -49.563, -93.149, 28.951, 56.324, -17.053]
  Call Extruder(25640.20666)
  MoveL 2731 to (-5.96, 26.09, 120) mm, rotated rx 180 ry 0 rz 180 deg; joints [-155.969, -49.176, -94.16, 29.067, 56.951, -16.864]
  Call Extruder(25649.57145)
  MoveL 2732 to (-11.61, 24.12, 120) mm, rotated rx 180 ry 0 rz 180 deg; joints [-155.891, -48.78, -95.208, 28.953, 57.543, -16.536]
  Call Extruder(25658.93637)
  MoveL 2733 to (-16.69, 20.93, 120) mm, rotated rx 180 ry 0 rz -180 deg; joints [-156.025, -48.394, -96.241, 28.605, 58.072, -16.087]
  Call Extruder(25668.30158)
  MoveL 2734 to (-20.93, 16.69, 120) mm, rotated rx -180 ry 0 rz 180 deg; joints [-156.374, -48.038, -97.206, 28.032, 58.514, -15.54]
  Call Extruder(25677.66649)
  MoveL 2735 to (-24.11, 11.61, 120) mm, rotated rx 180 ry 0 rz 180 deg; joints [-156.928, -47.729, -98.054, 27.254, 58.846, -14.922]
  Call Extruder(25687.03129)
  MoveL 2736 to (-26.09, 5.96, 120) mm, rotated rx -180 ry 0 rz 180 deg; joints [-157.665, -47.483, -98.738, 26.303, 59.051, -14.262]
  Call Extruder(25696.39640)
  MoveL 2737 to (-26.77, 0, 120) mm, rotated rx 180 ry 0 rz 180 deg; joints [-158.546, -47.31, -99.222, 25.225, 59.119, -13.593]
  Call Extruder(25701.18514)
  MoveL 2738 to (-26.42, -3.05, 120) mm, rotated rx -180 ry 0 rz 180 deg; joints [-159.044, -47.263, -99.354, 24.639, 59.081, -13.261]
  Set speed (130.0 mm/s)
  MoveL 2739 to (-41.86, -6.3, 120) mm, rotated rx 180 ry 0 rz 180 deg; joints [-158.606, -46.353, -101.97, 24.72, 60.729, -12.685]
  Call Extruder(25706.18298)
  Set speed (60.0 mm/s)
  MoveL 2740 to (-41.51, -9.47, 120) mm, rotated rx 180 ry 0 rz 180 deg; joints [-159.151, -46.308, -102.105, 24.088, 60.692, -12.344]
  Call Extruder(25721.07863)
  MoveL 2741 to (-38.36, -18.47, 120) mm, rotated rx 180 ry 0 rz 180 deg; joints [-160.835, -46.301, -102.125, 22.192, 60.357, -11.407]
  Call Extruder(25735.97448)
  MoveL 2742 to (-33.28, -26.54, 120) mm, rotated rx -180 ry 0 rz 180 deg; joints [-162.466, -46.429, -101.746, 20.398, 59.814, -10.591]
  Call Extruder(25750.87030)
  MoveL 2743 to (-26.54, -33.28, 120) mm, rotated rx 180 ry 0 rz -180 deg; joints [-163.93, -46.688, -100.994, 18.823, 59.087, -9.933]
  Call Extruder(25765.76615)
  MoveL 2744 to (-18.47, -38.36, 120) mm, rotated rx -180 ry 0 rz 180 deg; joints [-165.137, -47.066, -99.913, 17.564, 58.216, -9.465]
  Call Extruder(25780.66180)
  MoveL 2745 to (-9.47, -41.51, 120) mm, rotated rx 180 ry 0 rz 180 deg; joints [-166.024, -47.544, -98.567, 16.689, 57.243, -9.214]
  Call Extruder(25795.55768)
  MoveL 2746 to (0, -42.57, 120) mm, rotated rx -180 ry 0 rz 180 deg; joints [-166.562, -48.102, -97.032, 16.236, 56.22, -9.197]
  Call Extruder(25807.92576)
  MoveL 2747 to (7.87, -41.69, 120) mm, rotated rx -180 ry 0 rz -180 deg; joints [-166.715, -48.606, -95.671, 16.217, 55.373, -9.384]
  Call Extruder(25810.45355)
  MoveL 2748 to (9.47, -41.51, 120) mm, rotated rx 180 ry 0 rz 180 deg; joints [-166.745, -48.711, -95.391, 16.214, 55.199, -9.423]
  Call Extruder(25825.34921)
  MoveL 2749 to (18.47, -38.36, 120) mm, rotated rx 180 ry 0 rz 180 deg; joints [-166.591, -49.342, -93.726, 16.606, 54.233, -9.888]
  Call Extruder(25840.24506)
  MoveL 2750 to (26.54, -33.28, 120) mm, rotated rx 180 ry 0 rz 180 deg; joints [-166.133, -49.962, -92.119, 17.377, 53.37, -10.576]
  Call Extruder(25855.14087)
  MoveL 2751 to (33.28, -26.54, 120) mm, rotated rx 180 ry 0 rz 180 deg; joints [-165.409, -50.539, -90.646, 18.473, 52.656, -11.456]
  Call Extruder(25870.03673)
  MoveL 2752 to (38.36, -18.47, 120) mm, rotated rx 180 ry 0 rz 180 deg; joints [-164.468, -51.044, -89.374, 19.83, 52.127, -12.483]
  Call Extruder(25884.93238)
  MoveL 2753 to (41.51, -9.47, 120) mm, rotated rx -180 ry 0 rz 180 deg; joints [-163.355, -51.45, -88.361, 21.374, 51.81, -13.602]
  Call Extruder(25899.82825)
  MoveL 2754 to (42.57, 0, 120) mm, rotated rx 180 ry 0 rz 180 deg; joints [-162.12, -51.736, -87.654, 23.024, 51.722, -14.749]
  Call Extruder(25914.72413)
  MoveL 2755 to (41.5, 9.47, 120) mm, rotated rx -180 ry 0 rz 180 deg; joints [-160.81, -51.887, -87.283, 24.701, 51.866, -15.856]
  Call Extruder(25929.61979)
  MoveL 2756 to (38.36, 18.47, 120) mm, rotated rx 180 ry 0 rz -180 deg; joints [-159.475, -51.894, -87.265, 26.33, 52.233, -16.862]
  Call Extruder(25944.51563)
  MoveL 2757 to (33.29, 26.54, 120) mm, rotated rx 180 ry 0 rz 180 deg; joints [-158.16, -51.757, -87.601, 27.841, 52.802, -17.709]
  Call Extruder(25959.41146)
  MoveL 2758 to (26.54, 33.29, 120) mm, rotated rx 180 ry 0 rz 180 deg; joints [-156.916, -51.484, -88.277, 29.176, 53.54, -18.356]
  Call Extruder(25974.30730)
  MoveL 2759 to (18.47, 38.36, 120) mm, rotated rx 180 ry 0 rz -180 deg; joints [-155.789, -51.089, -89.261, 30.285, 54.411, -18.771]
  Call Extruder(25989.20296)
  MoveL 2760 to (9.47, 41.51, 120) mm, rotated rx 180 ry 0 rz 180 deg; joints [-154.828, -50.593, -90.509, 31.126, 55.368, -18.941]
  Call Extruder(26004.09884)
  MoveL 2761 to (0, 42.57, 120) mm, rotated rx -180 ry 0 rz 180 deg; joints [-154.081, -50.021, -91.966, 31.668, 56.365, -18.863]
  Call Extruder(26018.99471)
  MoveL 2762 to (-9.47, 41.51, 120) mm, rotated rx -180 ry 0 rz 180 deg; joints [-153.594, -49.404, -93.563, 31.881, 57.355, -18.548]
  Call Extruder(26033.89036)
  MoveL 2763 to (-18.47, 38.36, 120) mm, rotated rx 180 ry 0 rz 180 deg; joints [-153.408, -48.773, -95.225, 31.748, 58.29, -18.016]
  Call Extruder(26048.78621)
  MoveL 2764 to (-26.54, 33.29, 120) mm, rotated rx 180 ry 0 rz 180 deg; joints [-153.557, -48.161, -96.873, 31.253, 59.127, -17.298]
  Call Extruder(26063.68203)
  MoveL 2765 to (-33.29, 26.54, 120) mm, rotated rx -180 ry 0 rz 180 deg; joints [-154.059, -47.597, -98.422, 30.398, 59.827, -16.428]
  Call Extruder(26078.57788)
  MoveL 2766 to (-38.36, 18.47, 120) mm, rotated rx 180 ry 0 rz 180 deg; joints [-154.913, -47.109, -99.79, 29.199, 60.356, -15.452]
  Call Extruder(26093.47354)
  MoveL 2767 to (-41.5, 9.47, 120) mm, rotated rx -180 ry 0 rz 180 deg; joints [-156.091, -46.721, -100.9, 27.697, 60.688, -14.413]
  Call Extruder(26108.36942)
  MoveL 2768 to (-42.57, 0, 120) mm, rotated rx 180 ry 0 rz -180 deg; joints [-157.533, -46.449, -101.688, 25.962, 60.803, -13.362]
  Call Extruder(26115.92370)
  MoveL 2769 to (-42.03, -4.8, 120) mm, rotated rx -180 ry 0 rz 180 deg; joints [-158.35, -46.375, -101.905, 25.015, 60.747, -12.845]
  Set speed (130.0 mm/s)
  MoveL 2770 to (-54.1, -7.67, 120) mm, rotated rx 180 ry 0 rz -180 deg; joints [-158.024, -45.698, -103.934, 25.066, 62.042, -12.368]
  Call Extruder(26119.99632)
  Set speed (30.0 mm/s)
  MoveL 2771 to (-53.59, -12.23, 120) mm, rotated rx 180 ry 0 rz -180 deg; joints [-158.835, -45.634, -104.13, 24.139, 61.992, -11.884]
  Call Extruder(26130.92646)
  MoveL 2772 to (-49.53, -23.85, 120) mm, rotated rx 180 ry 0 rz 180 deg; joints [-161.095, -45.625, -104.157, 21.62, 61.566, -10.687]
  Call Extruder(26141.85674)
  MoveL 2773 to (-42.98, -34.27, 120) mm, rotated rx -180 ry 0 rz 180 deg; joints [-163.275, -45.789, -103.656, 19.236, 60.866, -9.642]
  Call Extruder(26152.78686)
  MoveL 2774 to (-34.27, -42.98, 120) mm, rotated rx -180 ry 0 rz 180 deg; joints [-165.21, -46.119, -102.664, 17.157, 59.926, -8.794]
  Call Extruder(26163.71714)
  MoveL 2775 to (-23.85, -49.52, 120) mm, rotated rx 180 ry 0 rz 180 deg; joints [-166.774, -46.601, -101.245, 15.515, 58.797, -8.184]
  Call Extruder(26174.64728)
  MoveL 2776 to (-12.23, -53.59, 120) mm, rotated rx -180 ry 0 rz 180 deg; joints [-167.889, -47.216, -99.487, 14.399, 57.537, -7.846]
  Call Extruder(26185.57750)
  MoveL 2777 to (0, -54.97, 120) mm, rotated rx 180 ry 0 rz 180 deg; joints [-168.526, -47.934, -97.493, 13.848, 56.211, -7.806]
  Call Extruder(26193.83885)
  MoveL 2778 to (9.25, -53.93, 120) mm, rotated rx 180 ry 0 rz 180 deg; joints [-168.656, -48.524, -95.891, 13.857, 55.212, -8.011]
  Call Extruder(26196.50772)
  MoveL 2779 to (12.23, -53.59, 120) mm, rotated rx -180 ry 0 rz 180 deg; joints [-168.697, -48.72, -95.369, 13.863, 54.889, -8.079]
  Call Extruder(26207.43786)
  MoveL 2780 to (23.85, -49.53, 120) mm, rotated rx 180 ry 0 rz 180 deg; joints [-168.436, -49.534, -93.224, 14.414, 53.637, -8.664]
  Call Extruder(26218.36814)
  MoveL 2781 to (34.27, -42.98, 120) mm, rotated rx -180 ry 0 rz 180 deg; joints [-167.797, -50.337, -91.16, 15.448, 52.519, -9.545]
  Call Extruder(26229.29826)
  MoveL 2782 to (42.98, -34.27, 120) mm, rotated rx -180 ry 0 rz 180 deg; joints [-166.837, -51.085, -89.271, 16.894, 51.593, -10.685]
  Call Extruder(26240.22854)
  MoveL 2783 to (49.53, -23.85, 120) mm, rotated rx -180 ry 0 rz 180 deg; joints [-165.618, -51.74, -87.644, 18.665, 50.907, -12.025]
  Call Extruder(26251.15868)
  MoveL 2784 to (53.59, -12.23, 120) mm, rotated rx 180 ry 0 rz -180 deg; joints [-164.2, -52.267, -86.35, 20.663, 50.497, -13.491]
  Call Extruder(26262.08890)
  MoveL 2785 to (54.97, 0, 120) mm, rotated rx 180 ry 0 rz 180 deg; joints [-162.641, -52.639, -85.445, 22.787, 50.386, -14.995]
  Call Extruder(26273.01912)
  MoveL 2786 to (53.59, 12.23, 120) mm, rotated rx 180 ry 0 rz 180 deg; joints [-160.996, -52.835, -84.971, 24.932, 50.577, -16.447]
  Call Extruder(26283.94926)
  MoveL 2787 to (49.52, 23.85, 120) mm, rotated rx 180 ry 0 rz -180 deg; joints [-159.322, -52.844, -84.949, 27.001, 51.058, -17.758]
  Call Extruder(26294.87954)
  MoveL 2788 to (42.98, 34.27, 120) mm, rotated rx 180 ry 0 rz 180 deg; joints [-157.673, -52.666, -85.379, 28.909, 51.799, -18.856]
  Call Extruder(26305.80966)
  MoveL 2789 to (34.27, 42.98, 120) mm, rotated rx 180 ry 0 rz 180 deg; joints [-156.102, -52.312, -86.242, 30.589, 52.758, -19.684]
  Call Extruder(26316.73994)
  MoveL 2790 to (23.85, 49.52, 120) mm, rotated rx 180 ry 0 rz 180 deg; joints [-154.667, -51.798, -87.5, 31.982, 53.884, -20.206]
  Call Extruder(26327.67008)
  MoveL 2791 to (12.23, 53.59, 120) mm, rotated rx 180 ry 0 rz 180 deg; joints [-153.426, -51.155, -89.097, 33.047, 55.119, -20.407]
  Call Extruder(26338.60030)
  MoveL 2792 to (0, 54.97, 120) mm, rotated rx 180 ry 0 rz 180 deg; joints [-152.438, -50.414, -90.963, 33.746, 56.403, -20.288]
  Call Extruder(26349.53053)
  MoveL 2793 to (-12.23, 53.59, 120) mm, rotated rx 180 ry 0 rz -180 deg; joints [-151.764, -49.615, -93.014, 34.048, 57.673, -19.867]
  Call Extruder(26360.46066)
  MoveL 2794 to (-23.85, 49.52, 120) mm, rotated rx -180 ry 0 rz 180 deg; joints [-151.463, -48.8, -95.155, 33.922, 58.873, -19.17]
  Call Extruder(26371.39094)
  MoveL 2795 to (-34.27, 42.98, 120) mm, rotated rx -180 ry 0 rz 180 deg; joints [-151.589, -48.009, -97.286, 33.345, 59.948, -18.238]
  Call Extruder(26382.32106)
  MoveL 2796 to (-42.98, 34.27, 120) mm, rotated rx 180 ry 0 rz -180 deg; joints [-152.179, -47.283, -99.298, 32.302, 60.85, -17.117]
  Call Extruder(26393.25134)
  MoveL 2797 to (-49.53, 23.85, 120) mm, rotated rx 180 ry 0 rz 180 deg; joints [-153.248, -46.657, -101.084, 30.799, 61.535, -15.861]
  Call Extruder(26404.18149)
  MoveL 2798 to (-53.59, 12.23, 120) mm, rotated rx 180 ry 0 rz 180 deg; joints [-154.769, -46.16, -102.541, 28.876, 61.97, -14.529]
  Call Extruder(26415.11171)
  MoveL 2799 to (-54.97, 0, 120) mm, rotated rx 180 ry 0 rz -180 deg; joints [-156.673, -45.814, -103.579, 26.613, 62.127, -13.184]
  Call Extruder(26420.63733)
  MoveL 2800 to (-54.27, -6.18, 120) mm, rotated rx 180 ry 0 rz 180 deg; joints [-157.76, -45.72, -103.867, 25.368, 62.058, -12.526]
  Set speed (130.0 mm/s)
  MoveL 2801 to (-49.9, -9.51, 120) mm, rotated rx 180 ry 0 rz 180 deg; joints [-158.616, -45.873, -103.403, 24.489, 61.592, -12.227]
  MoveL 2802 to (2.97, -12.99, 120) mm, rotated rx 180 ry 0 rz -180 deg; joints [-162.152, -48.802, -95.151, 21.714, 55.934, -12.575]
  Call Extruder(26425.30090)
  Set speed (80.0 mm/s)
  MoveL 2803 to (5.78, -12.01, 120) mm, rotated rx 180 ry 0 rz 180 deg; joints [-162.141, -48.999, -94.628, 21.81, 55.635, -12.729]
  Call Extruder(26429.96452)
  MoveL 2804 to (8.31, -10.42, 120) mm, rotated rx -180 ry 0 rz -180 deg; joints [-162.027, -49.192, -94.119, 22.026, 55.367, -12.948]
  Call Extruder(26434.62871)
  MoveL 2805 to (10.42, -8.31, 120) mm, rotated rx -180 ry 0 rz -180 deg; joints [-161.819, -49.371, -93.65, 22.348, 55.145, -13.222]
  Call Extruder(26439.29234)
  MoveL 2806 to (12.01, -5.78, 120) mm, rotated rx 180 ry 0 rz 180 deg; joints [-161.529, -49.527, -93.242, 22.76, 54.981, -13.537]
  Call Extruder(26443.95591)
  MoveL 2807 to (12.99, -2.97, 120) mm, rotated rx 180 ry 0 rz -180 deg; joints [-161.171, -49.653, -92.916, 23.24, 54.881, -13.876]
  Call Extruder(26448.61986)
  MoveL 2808 to (13.33, 0, 120) mm, rotated rx 180 ry 0 rz -180 deg; joints [-160.763, -49.741, -92.688, 23.763, 54.851, -14.223]
  Call Extruder(26453.28381)
  MoveL 2809 to (13, 2.97, 120) mm, rotated rx 180 ry 0 rz 180 deg; joints [-160.324, -49.787, -92.568, 24.304, 54.893, -14.559]
  Call Extruder(26457.94739)
  MoveL 2810 to (12.01, 5.78, 120) mm, rotated rx -180 ry 0 rz -180 deg; joints [-159.874, -49.79, -92.562, 24.837, 55.005, -14.866]
  Call Extruder(26462.61102)
  MoveL 2811 to (10.42, 8.31, 120) mm, rotated rx 180 ry 0 rz 180 deg; joints [-159.432, -49.748, -92.671, 25.337, 55.179, -15.129]
  Call Extruder(26467.27521)
  MoveL 2812 to (8.31, 10.42, 120) mm, rotated rx 180 ry 0 rz 180 deg; joints [-159.021, -49.663, -92.889, 25.78, 55.408, -15.334]
  Call Extruder(26471.93883)
  MoveL 2813 to (5.78, 12.01, 120) mm, rotated rx -180 ry 0 rz 180 deg; joints [-158.657, -49.541, -93.206, 26.147, 55.68, -15.471]
  Call Extruder(26476.60240)
  MoveL 2814 to (2.97, 13, 120) mm, rotated rx 180 ry 0 rz 180 deg; joints [-158.359, -49.388, -93.606, 26.419, 55.98, -15.534]
  Call Extruder(26481.26636)
  MoveL 2815 to (0, 13.33, 120) mm, rotated rx 180 ry 0 rz 180 deg; joints [-158.143, -49.21, -94.071, 26.585, 56.295, -15.52]
  Call Extruder(26485.93031)
  MoveL 2816 to (-2.97, 12.99, 120) mm, rotated rx -180 ry 0 rz -180 deg; joints [-158.019, -49.018, -94.576, 26.634, 56.609, -15.43]
  Call Extruder(26490.59387)
  MoveL 2817 to (-5.78, 12.01, 120) mm, rotated rx 180 ry 0 rz -180 deg; joints [-157.997, -48.821, -95.099, 26.564, 56.905, -15.27]
  Call Extruder(26495.25750)
  MoveL 2818 to (-8.31, 10.42, 120) mm, rotated rx 180 ry 0 rz 180 deg; joints [-158.08, -48.629, -95.612, 26.376, 57.171, -15.048]
  Call Extruder(26499.92170)
  MoveL 2819 to (-10.42, 8.31, 120) mm, rotated rx 180 ry 0 rz 180 deg; joints [-158.266, -48.451, -96.089, 26.077, 57.391, -14.775]
  Call Extruder(26504.58532)
  MoveL 2820 to (-12.01, 5.78, 120) mm, rotated rx 180 ry 0 rz 180 deg; joints [-158.549, -48.296, -96.506, 25.68, 57.556, -14.465]
  Call Extruder(26509.24889)
  MoveL 2821 to (-13, 2.97, 120) mm, rotated rx 180 ry 0 rz -180 deg; joints [-158.913, -48.172, -96.841, 25.204, 57.657, -14.133]
  Call Extruder(26513.91285)
  MoveL 2822 to (-13.33, 0, 120) mm, rotated rx 180 ry 0 rz 180 deg; joints [-159.341, -48.085, -97.078, 24.673, 57.689, -13.795]
  Call Extruder(26518.57680)
  MoveL 2823 to (-12.99, -2.97, 120) mm, rotated rx 180 ry 0 rz 180 deg; joints [-159.811, -48.04, -97.202, 24.113, 57.65, -13.468]
  Call Extruder(26523.24037)
  MoveL 2824 to (-12.01, -5.78, 120) mm, rotated rx 180 ry 0 rz 180 deg; joints [-160.294, -48.038, -97.208, 23.554, 57.542, -13.168]
  Call Extruder(26527.90400)
  MoveL 2825 to (-10.42, -8.31, 120) mm, rotated rx -180 ry 0 rz -180 deg; joints [-160.766, -48.079, -97.095, 23.026, 57.37, -12.908]
  Call Extruder(26532.56818)
  MoveL 2826 to (-8.31, -10.42, 120) mm, rotated rx 180 ry 0 rz 180 deg; joints [-161.2, -48.162, -96.87, 22.56, 57.143, -12.702]
  Call Extruder(26537.23182)
  MoveL 2827 to (-5.78, -12.01, 120) mm, rotated rx 180 ry 0 rz 180 deg; joints [-161.572, -48.282, -96.543, 22.178, 56.871, -12.56]
  Call Extruder(26541.89538)
  MoveL 2828 to (-2.97, -12.99, 120) mm, rotated rx 180 ry 0 rz 180 deg; joints [-161.863, -48.434, -96.133, 21.902, 56.569, -12.489]
  Call Extruder(26546.55933)
  MoveL 2829 to (0, -13.33, 120) mm, rotated rx -180 ry 0 rz -180 deg; joints [-162.059, -48.61, -95.661, 21.745, 56.251, -12.494]
  Call Extruder(26551.22329)
  MoveL 2830 to (2.97, -12.99, 120) mm, rotated rx 180 ry 0 rz -180 deg; joints [-162.152, -48.802, -95.151, 21.714, 55.934, -12.575]
  Set speed (130.0 mm/s)
  MoveL 2831 to (2.97, -12.99, 125) mm, rotated rx -180 ry 0 rz -180 deg; joints [-162.152, -48.047, -95.424, 21.836, 55.487, -12.791]
  MoveL 2832 to (-26.25, -4.54, 125) mm, rotated rx -180 ry 0 rz 180 deg; joints [-159.288, -46.45, -99.698, 24.479, 58.598, -13.345]
  Call Extruder(26553.45591)
  Set speed (60.0 mm/s)
  MoveL 2833 to (-26.09, -5.96, 125) mm, rotated rx 180 ry 0 rz -180 deg; joints [-159.522, -46.429, -99.758, 24.203, 58.579, -13.188]
  Call Extruder(26562.82070)
  MoveL 2834 to (-24.11, -11.61, 125) mm, rotated rx 180 ry 0 rz 180 deg; joints [-160.532, -46.424, -99.77, 23.046, 58.361, -12.58]
  Call Extruder(26572.18562)
  MoveL 2835 to (-20.93, -16.69, 125) mm, rotated rx 180 ry 0 rz 180 deg; joints [-161.513, -46.508, -99.538, 21.953, 58.015, -12.052]
  Call Extruder(26581.55082)
  MoveL 2836 to (-16.69, -20.93, 125) mm, rotated rx 180 ry 0 rz 180 deg; joints [-162.406, -46.677, -99.075, 20.987, 57.558, -11.628]
  Call Extruder(26590.91574)
  MoveL 2837 to (-11.61, -24.12, 125) mm, rotated rx 180 ry 0 rz 180 deg; joints [-163.159, -46.923, -98.408, 20.205, 57.014, -11.33]
  Call Extruder(26600.28053)
  MoveL 2838 to (-5.96, -26.09, 125) mm, rotated rx 180 ry 0 rz 180 deg; joints [-163.733, -47.233, -97.573, 19.65, 56.408, -11.175]
  Call Extruder(26609.64564)
  MoveL 2839 to (0, -26.77, 125) mm, rotated rx 180 ry 0 rz 180 deg; joints [-164.103, -47.593, -96.615, 19.346, 55.773, -11.171]
  Call Extruder(26619.01075)
  MoveL 2840 to (5.96, -26.09, 125) mm, rotated rx -180 ry 0 rz 180 deg; joints [-164.258, -47.985, -95.585, 19.307, 55.141, -11.323]
  Call Extruder(26628.37555)
  MoveL 2841 to (11.61, -24.12, 125) mm, rotated rx 180 ry 0 rz 180 deg; joints [-164.201, -48.389, -94.535, 19.527, 54.543, -11.625]
  Call Extruder(26637.74046)
  MoveL 2842 to (16.69, -20.93, 125) mm, rotated rx 180 ry 0 rz 180 deg; joints [-163.944, -48.786, -93.517, 19.988, 54.01, -12.065]
  Call Extruder(26647.10566)
  MoveL 2843 to (20.93, -16.69, 125) mm, rotated rx 180 ry 0 rz 180 deg; joints [-163.508, -49.154, -92.581, 20.661, 53.571, -12.622]
  Call Extruder(26656.47059)
  MoveL 2844 to (24.12, -11.61, 125) mm, rotated rx 180 ry 0 rz 180 deg; joints [-162.92, -49.475, -91.77, 21.505, 53.246, -13.267]
  Call Extruder(26665.83538)
  MoveL 2845 to (26.09, -5.96, 125) mm, rotated rx 180 ry 0 rz -180 deg; joints [-162.209, -49.733, -91.124, 22.477, 53.053, -13.966]
  Call Extruder(26675.20048)
  MoveL 2846 to (26.77, 0, 125) mm, rotated rx 180 ry 0 rz -180 deg; joints [-161.41, -49.914, -90.671, 23.526, 53.001, -14.681]
  Call Extruder(26684.56558)
  MoveL 2847 to (26.09, 5.96, 125) mm, rotated rx 180 ry 0 rz 180 deg; joints [-160.556, -50.01, -90.434, 24.601, 53.093, -15.374]
  Call Extruder(26693.93039)
  MoveL 2848 to (24.11, 11.61, 125) mm, rotated rx -180 ry 0 rz 180 deg; joints [-159.683, -50.014, -90.423, 25.653, 53.323, -16.006]
  Call Extruder(26703.29530)
  MoveL 2849 to (20.93, 16.69, 125) mm, rotated rx 180 ry 0 rz 180 deg; joints [-158.826, -49.928, -90.638, 26.635, 53.679, -16.545]
  Call Extruder(26712.66051)
  MoveL 2850 to (16.69, 20.93, 125) mm, rotated rx 180 ry 0 rz 180 deg; joints [-158.019, -49.754, -91.07, 27.505, 54.142, -16.962]
  Call Extruder(26722.02542)
  MoveL 2851 to (11.61, 24.12, 125) mm, rotated rx -180 ry 0 rz 180 deg; joints [-157.299, -49.504, -91.698, 28.225, 54.687, -17.238]
  Call Extruder(26731.39022)
  MoveL 2852 to (5.96, 26.09, 125) mm, rotated rx 180 ry 0 rz 180 deg; joints [-156.697, -49.188, -92.494, 28.766, 55.288, -17.361]
  Call Extruder(26740.75533)
  MoveL 2853 to (0, 26.77, 125) mm, rotated rx 180 ry 0 rz -180 deg; joints [-156.245, -48.824, -93.42, 29.104, 55.914, -17.327]
  Call Extruder(26750.12043)
  MoveL 2854 to (-5.96, 26.09, 125) mm, rotated rx -180 ry 0 rz 180 deg; joints [-155.969, -48.429, -94.432, 29.219, 56.536, -17.141]
  Call Extruder(26759.48523)
  MoveL 2855 to (-11.61, 24.11, 125) mm, rotated rx -180 ry 0 rz 180 deg; joints [-155.891, -48.025, -95.481, 29.103, 57.122, -16.814]
  Call Extruder(26768.85014)
  MoveL 2856 to (-16.69, 20.93, 125) mm, rotated rx 180 ry 0 rz -180 deg; joints [-156.025, -47.631, -96.516, 28.752, 57.644, -16.364]
  Call Extruder(26778.21535)
  MoveL 2857 to (-20.93, 16.69, 125) mm, rotated rx 180 ry 0 rz 180 deg; joints [-156.374, -47.267, -97.483, 28.176, 58.078, -15.814]
  Call Extruder(26787.58026)
  MoveL 2858 to (-24.11, 11.61, 125) mm, rotated rx 180 ry 0 rz 180 deg; joints [-156.928, -46.951, -98.332, 27.394, 58.401, -15.191]
  Call Extruder(26796.94507)
  MoveL 2859 to (-26.09, 5.96, 125) mm, rotated rx -180 ry 0 rz 180 deg; joints [-157.665, -46.698, -99.018, 26.438, 58.599, -14.525]
  Call Extruder(26806.31017)
  MoveL 2860 to (-26.77, 0, 125) mm, rotated rx -180 ry 0 rz 180 deg; joints [-158.546, -46.521, -99.502, 25.356, 58.659, -13.846]
  Call Extruder(26811.09891)
  MoveL 2861 to (-26.42, -3.05, 125) mm, rotated rx 180 ry 0 rz 180 deg; joints [-159.044, -46.473, -99.635, 24.767, 58.618, -13.51]
  Set speed (130.0 mm/s)
  MoveL 2862 to (-41.86, -6.3, 125) mm, rotated rx 180 ry 0 rz 180 deg; joints [-158.606, -45.539, -102.256, 24.845, 60.249, -12.94]
  Call Extruder(26816.09675)
  Set speed (60.0 mm/s)
  MoveL 2863 to (-41.5, -9.47, 125) mm, rotated rx 180 ry 0 rz -180 deg; joints [-159.151, -45.492, -102.391, 24.211, 60.209, -12.593]
  Call Extruder(26830.99240)
  MoveL 2864 to (-38.36, -18.47, 125) mm, rotated rx -180 ry 0 rz 180 deg; joints [-160.835, -45.485, -102.411, 22.307, 59.867, -11.638]
  Call Extruder(26845.88825)
  MoveL 2865 to (-33.28, -26.54, 125) mm, rotated rx 180 ry 0 rz 180 deg; joints [-162.466, -45.617, -102.032, 20.506, 59.32, -10.804]
  Call Extruder(26860.78407)
  MoveL 2866 to (-26.54, -33.28, 125) mm, rotated rx -180 ry 0 rz -180 deg; joints [-163.93, -45.883, -101.278, 18.925, 58.594, -10.13]
  Call Extruder(26875.67992)
  MoveL 2867 to (-18.47, -38.36, 125) mm, rotated rx -180 ry 0 rz 180 deg; joints [-165.137, -46.271, -100.194, 17.661, 57.726, -9.649]
  Call Extruder(26890.57557)
  MoveL 2868 to (-9.47, -41.5, 125) mm, rotated rx 180 ry 0 rz 180 deg; joints [-166.024, -46.762, -98.846, 16.783, 56.761, -9.387]
  Call Extruder(26905.47145)
  MoveL 2869 to (0, -42.57, 125) mm, rotated rx 180 ry 0 rz 180 deg; joints [-166.562, -47.332, -97.309, 16.33, 55.747, -9.364]
  Call Extruder(26918.58282)
  MoveL 2870 to (8.34, -41.63, 125) mm, rotated rx 180 ry 0 rz 180 deg; joints [-166.724, -47.879, -95.862, 16.31, 54.857, -9.561]
  Call Extruder(26920.36733)
  MoveL 2871 to (9.47, -41.5, 125) mm, rotated rx 180 ry 0 rz 180 deg; joints [-166.745, -47.955, -95.664, 16.309, 54.736, -9.588]
  Call Extruder(26935.26298)
  MoveL 2872 to (18.47, -38.36, 125) mm, rotated rx 180 ry 0 rz 180 deg; joints [-166.591, -48.598, -93.997, 16.705, 53.78, -10.056]
  Call Extruder(26950.15883)
  MoveL 2873 to (26.54, -33.28, 125) mm, rotated rx 180 ry 0 rz 180 deg; joints [-166.133, -49.23, -92.388, 17.481, 52.929, -10.749]
  Call Extruder(26965.05465)
  MoveL 2874 to (33.29, -26.54, 125) mm, rotated rx 180 ry 0 rz 180 deg; joints [-165.409, -49.817, -90.913, 18.585, 52.225, -11.638]
  Call Extruder(26979.95050)
  MoveL 2875 to (38.36, -18.47, 125) mm, rotated rx 180 ry 0 rz 180 deg; joints [-164.468, -50.331, -89.64, 19.95, 51.706, -12.677]
  Call Extruder(26994.84615)
  MoveL 2876 to (41.5, -9.47, 125) mm, rotated rx 180 ry 0 rz 180 deg; joints [-163.355, -50.743, -88.626, 21.501, 51.399, -13.808]
  Call Extruder(27009.74203)
  MoveL 2877 to (42.57, 0, 125) mm, rotated rx 180 ry 0 rz 180 deg; joints [-162.12, -51.034, -87.918, 23.16, 51.319, -14.968]
  Call Extruder(27024.63790)
  MoveL 2878 to (41.5, 9.47, 125) mm, rotated rx -180 ry 0 rz 180 deg; joints [-160.81, -51.186, -87.547, 24.845, 51.47, -16.089]
  Call Extruder(27039.53356)
  MoveL 2879 to (38.36, 18.47, 125) mm, rotated rx -180 ry 0 rz 180 deg; joints [-159.475, -51.194, -87.529, 26.481, 51.843, -17.107]
  Call Extruder(27054.42941)
  MoveL 2880 to (33.29, 26.54, 125) mm, rotated rx 180 ry 0 rz -180 deg; joints [-158.16, -51.055, -87.866, 27.998, 52.415, -17.967]
  Call Extruder(27069.32523)
  MoveL 2881 to (26.54, 33.28, 125) mm, rotated rx 180 ry 0 rz 180 deg; joints [-156.916, -50.778, -88.542, 29.337, 53.155, -18.624]
  Call Extruder(27084.22107)
  MoveL 2882 to (18.47, 38.36, 125) mm, rotated rx 180 ry 0 rz -180 deg; joints [-155.789, -50.377, -89.527, 30.448, 54.025, -19.05]
  Call Extruder(27099.11674)
  MoveL 2883 to (9.47, 41.51, 125) mm, rotated rx -180 ry 0 rz 180 deg; joints [-154.828, -49.872, -90.777, 31.29, 54.98, -19.227]
  Call Extruder(27114.01261)
  MoveL 2884 to (0, 42.57, 125) mm, rotated rx 180 ry 0 rz 180 deg; joints [-154.081, -49.291, -92.234, 31.831, 55.972, -19.156]
  Call Extruder(27128.90848)
  MoveL 2885 to (-9.47, 41.51, 125) mm, rotated rx 180 ry 0 rz 180 deg; joints [-153.594, -48.662, -93.834, 32.043, 56.955, -18.845]
  Call Extruder(27143.80414)
  MoveL 2886 to (-18.47, 38.36, 125) mm, rotated rx -180 ry 0 rz -180 deg; joints [-153.408, -48.018, -95.499, 31.906, 57.88, -18.316]
  Call Extruder(27158.69999)
  MoveL 2887 to (-26.54, 33.28, 125) mm, rotated rx 180 ry 0 rz 180 deg; joints [-153.557, -47.392, -97.149, 31.407, 58.706, -17.596]
  Call Extruder(27173.59580)
  MoveL 2888 to (-33.28, 26.54, 125) mm, rotated rx 180 ry 0 rz 180 deg; joints [-154.059, -46.815, -98.701, 30.547, 59.394, -16.724]
  Call Extruder(27188.49165)
  MoveL 2889 to (-38.36, 18.47, 125) mm, rotated rx 180 ry 0 rz -180 deg; joints [-154.913, -46.315, -100.071, 29.343, 59.909, -15.74]
  Call Extruder(27203.38731)
  MoveL 2890 to (-41.5, 9.47, 125) mm, rotated rx -180 ry 0 rz -180 deg; joints [-156.091, -45.917, -101.184, 27.835, 60.227, -14.692]
  Call Extruder(27218.28318)
  MoveL 2891 to (-42.57, 0, 125) mm, rotated rx -180 ry 0 rz -180 deg; joints [-157.533, -45.638, -101.973, 26.092, 60.33, -13.627]
  Call Extruder(27225.83747)
  MoveL 2892 to (-42.03, -4.8, 125) mm, rotated rx 180 ry 0 rz 180 deg; joints [-158.35, -45.562, -102.191, 25.142, 60.269, -13.102]
  Set speed (130.0 mm/s)
  MoveL 2893 to (-54.1, -7.67, 125) mm, rotated rx -180 ry 0 rz 180 deg; joints [-158.024, -44.864, -104.225, 25.19, 61.55, -12.63]
  Call Extruder(27229.91010)
  Set speed (30.0 mm/s)
  MoveL 2894 to (-53.59, -12.23, 125) mm, rotated rx -180 ry 0 rz 180 deg; joints [-158.835, -44.797, -104.422, 24.259, 61.495, -12.138]
  Call Extruder(27240.84023)
  MoveL 2895 to (-49.52, -23.85, 125) mm, rotated rx -180 ry 0 rz 180 deg; joints [-161.095, -44.788, -104.448, 21.73, 61.059, -10.916]
  Call Extruder(27251.77052)
  MoveL 2896 to (-42.98, -34.27, 125) mm, rotated rx 180 ry 0 rz 180 deg; joints [-163.275, -44.957, -103.947, 19.337, 60.355, -9.847]
  Call Extruder(27262.70063)
  MoveL 2897 to (-34.27, -42.98, 125) mm, rotated rx 180 ry 0 rz 180 deg; joints [-165.21, -45.297, -102.952, 17.249, 59.417, -8.977]
  Call Extruder(27273.63092)
  MoveL 2898 to (-23.85, -49.53, 125) mm, rotated rx -180 ry 0 rz 180 deg; joints [-166.774, -45.794, -101.529, 15.601, 58.293, -8.349]
  Call Extruder(27284.56105)
  MoveL 2899 to (-12.23, -53.59, 125) mm, rotated rx -180 ry 0 rz 180 deg; joints [-167.889, -46.425, -99.768, 14.48, 57.043, -7.997]
  Call Extruder(27295.49127)
  MoveL 2900 to (0, -54.97, 125) mm, rotated rx 180 ry 0 rz 180 deg; joints [-168.526, -47.16, -97.77, 13.928, 55.729, -7.95]
  Call Extruder(27304.17504)
  MoveL 2901 to (9.72, -53.87, 125) mm, rotated rx -180 ry 0 rz 180 deg; joints [-168.663, -47.795, -96.082, 13.94, 54.69, -8.164]
  Call Extruder(27306.42149)
  MoveL 2902 to (12.23, -53.59, 125) mm, rotated rx 180 ry 0 rz 180 deg; joints [-168.697, -47.963, -95.643, 13.945, 54.421, -8.221]
  Call Extruder(27317.35164)
  MoveL 2903 to (23.85, -49.53, 125) mm, rotated rx -180 ry 0 rz 180 deg; joints [-168.436, -48.794, -93.494, 14.501, 53.183, -8.81]
  Call Extruder(27328.28192)
  MoveL 2904 to (34.27, -42.98, 125) mm, rotated rx 180 ry 0 rz 180 deg; joints [-167.797, -49.611, -91.428, 15.543, 52.078, -9.7]
  Call Extruder(27339.21203)
  MoveL 2905 to (42.98, -34.27, 125) mm, rotated rx -180 ry 0 rz 180 deg; joints [-166.837, -50.372, -89.537, 16.998, 51.165, -10.851]
  Call Extruder(27350.14232)
  MoveL 2906 to (49.53, -23.85, 125) mm, rotated rx 180 ry 0 rz 180 deg; joints [-165.618, -51.038, -87.908, 18.78, 50.492, -12.206]
  Call Extruder(27361.07245)
  MoveL 2907 to (53.59, -12.23, 125) mm, rotated rx 180 ry 0 rz -180 deg; joints [-164.2, -51.573, -86.613, 20.79, 50.094, -13.689]
  Call Extruder(27372.00267)
  MoveL 2908 to (54.97, 0, 125) mm, rotated rx 180 ry 0 rz 180 deg; joints [-162.641, -51.95, -85.708, 22.925, 49.993, -15.211]
  Call Extruder(27382.93289)
  MoveL 2909 to (53.59, 12.23, 125) mm, rotated rx 180 ry 0 rz 180 deg; joints [-160.996, -52.148, -85.234, 25.08, 50.193, -16.679]
  Call Extruder(27393.86304)
  MoveL 2910 to (49.53, 23.85, 125) mm, rotated rx 180 ry 0 rz -180 deg; joints [-159.322, -52.158, -85.211, 27.158, 50.68, -18.007]
  Call Extruder(27404.79331)
  MoveL 2911 to (42.98, 34.27, 125) mm, rotated rx 180 ry 0 rz -180 deg; joints [-157.673, -51.977, -85.641, 29.073, 51.426, -19.12]
  Call Extruder(27415.72344)
  MoveL 2912 to (34.27, 42.98, 125) mm, rotated rx 180 ry 0 rz -180 deg; joints [-156.102, -51.618, -86.505, 30.757, 52.388, -19.961]
  Call Extruder(27426.65371)
  MoveL 2913 to (23.85, 49.52, 125) mm, rotated rx 180 ry 0 rz -180 deg; joints [-154.667, -51.097, -87.764, 32.153, 53.514, -20.494]
  Call Extruder(27437.58386)
  MoveL 2914 to (12.23, 53.59, 125) mm, rotated rx 180 ry 0 rz 180 deg; joints [-153.426, -50.443, -89.363, 33.218, 54.746, -20.705]
  Call Extruder(27448.51408)
  MoveL 2915 to (0, 54.97, 125) mm, rotated rx -180 ry 0 rz 180 deg; joints [-152.438, -49.69, -91.231, 33.916, 56.024, -20.594]
  Call Extruder(27459.44430)
  MoveL 2916 to (-12.23, 53.59, 125) mm, rotated rx 180 ry 0 rz 180 deg; joints [-151.764, -48.877, -93.284, 34.215, 57.286, -20.178]
  Call Extruder(27470.37444)
  MoveL 2917 to (-23.85, 49.52, 125) mm, rotated rx 180 ry 0 rz 180 deg; joints [-151.463, -48.045, -95.429, 34.086, 58.474, -19.485]
  Call Extruder(27481.30472)
  MoveL 2918 to (-34.27, 42.98, 125) mm, rotated rx 180 ry 0 rz 180 deg; joints [-151.589, -47.237, -97.563, 33.504, 59.535, -18.554]
  Call Extruder(27492.23484)
  MoveL 2919 to (-42.98, 34.27, 125) mm, rotated rx 180 ry 0 rz -180 deg; joints [-152.179, -46.494, -99.578, 32.456, 60.42, -17.429]
  Call Extruder(27503.16512)
  MoveL 2920 to (-49.52, 23.85, 125) mm, rotated rx 180 ry 0 rz 180 deg; joints [-153.248, -45.851, -101.368, 30.946, 61.088, -16.166]
  Call Extruder(27514.09526)
  MoveL 2921 to (-53.59, 12.23, 125) mm, rotated rx 180 ry 0 rz 180 deg; joints [-154.769, -45.34, -102.829, 29.014, 61.504, -14.822]
  Call Extruder(27525.02548)
  MoveL 2922 to (-54.97, 0, 125) mm, rotated rx 180 ry 0 rz -180 deg; joints [-156.673, -44.984, -103.869, 26.742, 61.643, -13.459]
  Call Extruder(27530.55110)
  MoveL 2923 to (-54.27, -6.18, 125) mm, rotated rx 180 ry 0 rz 180 deg; joints [-157.76, -44.886, -104.158, 25.493, 61.568, -12.791]
  Set speed (130.0 mm/s)
  MoveL 2924 to (-49.9, -9.51, 125) mm, rotated rx -180 ry 0 rz 180 deg; joints [-158.616, -45.044, -103.692, 24.612, 61.102, -12.482]
  MoveL 2925 to (2.97, -12.99, 125) mm, rotated rx -180 ry 0 rz -180 deg; joints [-162.152, -48.047, -95.424, 21.836, 55.487, -12.791]
  Call Extruder(27535.21467)
  Set speed (80.0 mm/s)
  MoveL 2926 to (5.78, -12.01, 125) mm, rotated rx -180 ry 0 rz 180 deg; joints [-162.141, -48.248, -94.9, 21.933, 55.191, -12.945]
  Call Extruder(27539.87829)
  MoveL 2927 to (8.31, -10.42, 125) mm, rotated rx 180 ry 0 rz -180 deg; joints [-162.027, -48.445, -94.391, 22.15, 54.927, -13.165]
  Call Extruder(27544.54248)
  MoveL 2928 to (10.42, -8.31, 125) mm, rotated rx 180 ry 0 rz 180 deg; joints [-161.819, -48.628, -93.921, 22.474, 54.709, -13.442]
  Call Extruder(27549.20612)
  MoveL 2929 to (12.01, -5.78, 125) mm, rotated rx -180 ry 0 rz 180 deg; joints [-161.529, -48.787, -93.512, 22.889, 54.548, -13.76]
  Call Extruder(27553.86968)
  MoveL 2930 to (13, -2.97, 125) mm, rotated rx 180 ry 0 rz -180 deg; joints [-161.171, -48.915, -93.186, 23.371, 54.451, -14.103]
  Call Extruder(27558.53364)
  MoveL 2931 to (13.33, 0, 125) mm, rotated rx 180 ry 0 rz 180 deg; joints [-160.763, -49.005, -92.958, 23.897, 54.425, -14.454]
  Call Extruder(27563.19759)
  MoveL 2932 to (13, 2.97, 125) mm, rotated rx 180 ry 0 rz -180 deg; joints [-160.324, -49.052, -92.838, 24.44, 54.469, -14.794]
  Call Extruder(27567.86116)
  MoveL 2933 to (12.01, 5.78, 125) mm, rotated rx 180 ry 0 rz -180 deg; joints [-159.874, -49.054, -92.832, 24.975, 54.582, -15.106]
  Call Extruder(27572.52479)
  MoveL 2934 to (10.42, 8.31, 125) mm, rotated rx 180 ry 0 rz 180 deg; joints [-159.432, -49.012, -92.941, 25.477, 54.758, -15.373]
  Call Extruder(27577.18898)
  MoveL 2935 to (8.31, 10.42, 125) mm, rotated rx -180 ry 0 rz 180 deg; joints [-159.021, -48.926, -93.159, 25.922, 54.987, -15.582]
  Call Extruder(27581.85260)
  MoveL 2936 to (5.78, 12.01, 125) mm, rotated rx 180 ry 0 rz 180 deg; joints [-158.657, -48.802, -93.476, 26.289, 55.259, -15.723]
  Call Extruder(27586.51618)
  MoveL 2937 to (2.97, 13, 125) mm, rotated rx 180 ry 0 rz 180 deg; joints [-158.359, -48.645, -93.877, 26.563, 55.558, -15.788]
  Call Extruder(27591.18013)
  MoveL 2938 to (0, 13.33, 125) mm, rotated rx -180 ry 0 rz 180 deg; joints [-158.143, -48.464, -94.342, 26.728, 55.871, -15.776]
  Call Extruder(27595.84409)
  MoveL 2939 to (-2.97, 12.99, 125) mm, rotated rx -180 ry 0 rz 180 deg; joints [-158.019, -48.268, -94.849, 26.777, 56.182, -15.688]
  Call Extruder(27600.50765)
  MoveL 2940 to (-5.78, 12.01, 125) mm, rotated rx -180 ry 0 rz 180 deg; joints [-157.997, -48.067, -95.372, 26.706, 56.475, -15.528]
  Call Extruder(27605.17128)
  MoveL 2941 to (-8.31, 10.42, 125) mm, rotated rx 180 ry 0 rz 180 deg; joints [-158.08, -47.87, -95.886, 26.516, 56.737, -15.305]
  Call Extruder(27609.83547)
  MoveL 2942 to (-10.42, 8.31, 125) mm, rotated rx -180 ry 0 rz 180 deg; joints [-158.266, -47.689, -96.363, 26.216, 56.954, -15.03]
  Call Extruder(27614.49910)
  MoveL 2943 to (-12.01, 5.78, 125) mm, rotated rx -180 ry 0 rz 180 deg; joints [-158.549, -47.531, -96.781, 25.817, 57.115, -14.718]
  Call Extruder(27619.16267)
  MoveL 2944 to (-12.99, 2.97, 125) mm, rotated rx 180 ry 0 rz -180 deg; joints [-158.913, -47.404, -97.117, 25.339, 57.212, -14.382]
  Call Extruder(27623.82662)
  MoveL 2945 to (-13.33, 0, 125) mm, rotated rx -180 ry 0 rz 180 deg; joints [-159.341, -47.315, -97.354, 24.804, 57.241, -14.041]
  Call Extruder(27628.49058)
  MoveL 2946 to (-12.99, -2.97, 125) mm, rotated rx 180 ry 0 rz 180 deg; joints [-159.811, -47.269, -97.479, 24.242, 57.199, -13.709]
  Call Extruder(27633.15414)
  MoveL 2947 to (-12.01, -5.78, 125) mm, rotated rx 180 ry 0 rz 180 deg; joints [-160.294, -47.266, -97.484, 23.681, 57.089, -13.403]
  Call Extruder(27637.81777)
  MoveL 2948 to (-10.42, -8.31, 125) mm, rotated rx -180 ry 0 rz 180 deg; joints [-160.766, -47.309, -97.371, 23.152, 56.916, -13.138]
  Call Extruder(27642.48196)
  MoveL 2949 to (-8.31, -10.42, 125) mm, rotated rx 180 ry 0 rz 180 deg; joints [-161.2, -47.393, -97.146, 22.683, 56.688, -12.928]
  Call Extruder(27647.14559)
  MoveL 2950 to (-5.78, -12.01, 125) mm, rotated rx 180 ry 0 rz 180 deg; joints [-161.572, -47.517, -96.819, 22.3, 56.417, -12.782]
  Call Extruder(27651.80916)
  MoveL 2951 to (-2.97, -13, 125) mm, rotated rx -180 ry 0 rz 180 deg; joints [-161.863, -47.672, -96.408, 22.023, 56.116, -12.708]
  Call Extruder(27656.47311)
  MoveL 2952 to (0, -13.33, 125) mm, rotated rx -180 ry 0 rz -180 deg; joints [-162.059, -47.852, -95.935, 21.866, 55.801, -12.711]
  Call Extruder(27661.13707)
  MoveL 2953 to (2.97, -12.99, 125) mm, rotated rx -180 ry 0 rz -180 deg; joints [-162.152, -48.047, -95.424, 21.836, 55.487, -12.791]
  Set speed (130.0 mm/s)
  MoveL 2954 to (2.97, -12.99, 130) mm, rotated rx 180 ry 0 rz -180 deg; joints [-162.152, -47.294, -95.687, 21.963, 55.034, -13.013]
  MoveL 2955 to (-26.25, -4.54, 130) mm, rotated rx 180 ry 0 rz 180 deg; joints [-159.288, -45.661, -99.969, 24.611, 58.126, -13.598]
  Call Extruder(27663.36969)
  Set speed (60.0 mm/s)
  MoveL 2956 to (-26.09, -5.96, 130) mm, rotated rx -180 ry 0 rz -180 deg; joints [-159.522, -45.639, -100.029, 24.335, 58.106, -13.438]
  Call Extruder(27672.73448)
  MoveL 2957 to (-24.11, -11.61, 130) mm, rotated rx 180 ry 0 rz 180 deg; joints [-160.532, -45.634, -100.041, 23.173, 57.884, -12.82]
  Call Extruder(27682.09940)
  MoveL 2958 to (-20.93, -16.69, 130) mm, rotated rx 180 ry 0 rz 180 deg; joints [-161.513, -45.721, -99.809, 22.075, 57.536, -12.281]
  Call Extruder(27691.46460)
  MoveL 2959 to (-16.69, -20.93, 130) mm, rotated rx 180 ry 0 rz 180 deg; joints [-162.406, -45.894, -99.345, 21.106, 57.079, -11.847]
  Call Extruder(27700.82953)
  MoveL 2960 to (-11.61, -24.12, 130) mm, rotated rx 180 ry 0 rz 180 deg; joints [-163.159, -46.145, -98.677, 20.321, 56.536, -11.541]
  Call Extruder(27710.19431)
  MoveL 2961 to (-5.96, -26.09, 130) mm, rotated rx 180 ry 0 rz 180 deg; joints [-163.733, -46.463, -97.84, 19.763, 55.935, -11.379]
  Call Extruder(27719.55942)
  MoveL 2962 to (0, -26.77, 130) mm, rotated rx -180 ry 0 rz 180 deg; joints [-164.103, -46.831, -96.881, 19.46, 55.305, -11.372]
  Call Extruder(27728.92452)
  MoveL 2963 to (5.96, -26.09, 130) mm, rotated rx 180 ry 0 rz 180 deg; joints [-164.258, -47.231, -95.849, 19.422, 54.678, -11.522]
  Call Extruder(27738.28933)
  MoveL 2964 to (11.61, -24.11, 130) mm, rotated rx 180 ry 0 rz 180 deg; joints [-164.201, -47.643, -94.798, 19.644, 54.087, -11.825]
  Call Extruder(27747.65424)
  MoveL 2965 to (16.69, -20.93, 130) mm, rotated rx 180 ry 0 rz 180 deg; joints [-163.944, -48.047, -93.778, 20.108, 53.562, -12.268]
  Call Extruder(27757.01945)
  MoveL 2966 to (20.93, -16.69, 130) mm, rotated rx 180 ry 0 rz 180 deg; joints [-163.508, -48.422, -92.84, 20.785, 53.13, -12.83]
  Call Extruder(27766.38437)
  MoveL 2967 to (24.11, -11.61, 130) mm, rotated rx -180 ry 0 rz 180 deg; joints [-162.92, -48.749, -92.029, 21.634, 52.812, -13.481]
  Call Extruder(27775.74916)
  MoveL 2968 to (26.09, -5.96, 130) mm, rotated rx -180 ry 0 rz -180 deg; joints [-162.209, -49.012, -91.382, 22.611, 52.625, -14.188]
  Call Extruder(27785.11426)
  MoveL 2969 to (26.77, 0, 130) mm, rotated rx 180 ry 0 rz -180 deg; joints [-161.41, -49.196, -90.929, 23.666, 52.579, -14.912]
  Call Extruder(27794.47937)
  MoveL 2970 to (26.09, 5.96, 130) mm, rotated rx 180 ry 0 rz 180 deg; joints [-160.556, -49.293, -90.692, 24.746, 52.676, -15.614]
  Call Extruder(27803.84417)
  MoveL 2971 to (24.12, 11.61, 130) mm, rotated rx 180 ry 0 rz -180 deg; joints [-159.683, -49.298, -90.68, 25.803, 52.91, -16.255]
  Call Extruder(27813.20908)
  MoveL 2972 to (20.93, 16.69, 130) mm, rotated rx 180 ry 0 rz 180 deg; joints [-158.826, -49.21, -90.896, 26.788, 53.268, -16.802]
  Call Extruder(27822.57429)
  MoveL 2973 to (16.69, 20.93, 130) mm, rotated rx 180 ry 0 rz 180 deg; joints [-158.019, -49.034, -91.328, 27.661, 53.732, -17.227]
  Call Extruder(27831.93920)
  MoveL 2974 to (11.61, 24.11, 130) mm, rotated rx -180 ry 0 rz 180 deg; joints [-157.299, -48.779, -91.957, 28.383, 54.277, -17.509]
  Call Extruder(27841.30400)
  MoveL 2975 to (5.96, 26.09, 130) mm, rotated rx 180 ry 0 rz -180 deg; joints [-156.697, -48.457, -92.753, 28.925, 54.875, -17.638]
  Call Extruder(27850.66911)
  MoveL 2976 to (0, 26.77, 130) mm, rotated rx -180 ry 0 rz -180 deg; joints [-156.245, -48.086, -93.681, 29.262, 55.498, -17.608]
  Call Extruder(27860.03421)
  MoveL 2977 to (-5.96, 26.09, 130) mm, rotated rx -180 ry 0 rz 180 deg; joints [-155.969, -47.684, -94.694, 29.377, 56.115, -17.425]
  Call Extruder(27869.39900)
  MoveL 2978 to (-11.61, 24.12, 130) mm, rotated rx 180 ry 0 rz 180 deg; joints [-155.891, -47.272, -95.745, 29.258, 56.694, -17.099]
  Call Extruder(27878.76392)
  MoveL 2979 to (-16.69, 20.93, 130) mm, rotated rx 180 ry 0 rz -180 deg; joints [-156.025, -46.869, -96.781, 28.905, 57.209, -16.648]
  Call Extruder(27888.12913)
  MoveL 2980 to (-20.93, 16.69, 130) mm, rotated rx 180 ry 0 rz -180 deg; joints [-156.374, -46.497, -97.75, 28.326, 57.635, -16.095]
  Call Extruder(27897.49404)
  MoveL 2981 to (-24.11, 11.61, 130) mm, rotated rx 180 ry 0 rz 180 deg; joints [-156.928, -46.174, -98.601, 27.539, 57.95, -15.467]
  Call Extruder(27906.85884)
  MoveL 2982 to (-26.09, 5.96, 130) mm, rotated rx 180 ry 0 rz -180 deg; joints [-157.665, -45.915, -99.288, 26.579, 58.139, -14.794]
  Call Extruder(27916.22395)
  MoveL 2983 to (-26.77, 0, 130) mm, rotated rx 180 ry 0 rz -180 deg; joints [-158.546, -45.734, -99.773, 25.492, 58.192, -14.107]
  Call Extruder(27921.01269)
  MoveL 2984 to (-26.42, -3.05, 130) mm, rotated rx -180 ry 0 rz 180 deg; joints [-159.044, -45.684, -99.906, 24.901, 58.148, -13.765]
  Set speed (130.0 mm/s)
  MoveL 2985 to (-41.86, -6.3, 130) mm, rotated rx -180 ry 0 rz 180 deg; joints [-158.606, -44.725, -102.533, 24.976, 59.762, -13.201]
  Call Extruder(27926.01053)
  Set speed (60.0 mm/s)
  MoveL 2986 to (-41.51, -9.47, 130) mm, rotated rx -180 ry 0 rz 180 deg; joints [-159.151, -44.677, -102.668, 24.339, 59.718, -12.849]
  Call Extruder(27940.90618)
  MoveL 2987 to (-38.36, -18.47, 130) mm, rotated rx 180 ry 0 rz 180 deg; joints [-160.835, -44.67, -102.688, 22.427, 59.37, -11.875]
  Call Extruder(27955.80203)
  MoveL 2988 to (-33.29, -26.54, 130) mm, rotated rx 180 ry 0 rz 180 deg; joints [-162.466, -44.806, -102.308, 20.619, 58.819, -11.023]
  Call Extruder(27970.69785)
  MoveL 2989 to (-26.54, -33.28, 130) mm, rotated rx 180 ry 0 rz -180 deg; joints [-163.93, -45.079, -101.552, 19.031, 58.094, -10.332]
  Call Extruder(27985.59371)
  MoveL 2990 to (-18.47, -38.36, 130) mm, rotated rx -180 ry 0 rz 180 deg; joints [-165.137, -45.477, -100.466, 17.762, 57.229, -9.837]
  Call Extruder(28000.48935)
  MoveL 2991 to (-9.47, -41.5, 130) mm, rotated rx 180 ry 0 rz 180 deg; joints [-166.024, -45.98, -99.115, 16.881, 56.27, -9.565]
  Call Extruder(28015.38523)
  MoveL 2992 to (0, -42.57, 130) mm, rotated rx 180 ry 0 rz 180 deg; joints [-166.562, -46.564, -97.575, 16.427, 55.265, -9.536]
  Call Extruder(28029.06537)
  MoveL 2993 to (8.7, -41.59, 130) mm, rotated rx 180 ry 0 rz 180 deg; joints [-166.731, -47.147, -96.064, 16.408, 54.347, -9.739]
  Call Extruder(28030.28109)
  MoveL 2994 to (9.47, -41.51, 130) mm, rotated rx -180 ry 0 rz 180 deg; joints [-166.745, -47.2, -95.929, 16.407, 54.265, -9.758]
  Call Extruder(28045.17676)
  MoveL 2995 to (18.47, -38.36, 130) mm, rotated rx 180 ry 0 rz 180 deg; joints [-166.591, -47.856, -94.259, 16.807, 53.321, -10.228]
  Call Extruder(28060.07261)
  MoveL 2996 to (26.54, -33.29, 130) mm, rotated rx -180 ry 0 rz -180 deg; joints [-166.133, -48.5, -92.647, 17.589, 52.48, -10.928]
  Call Extruder(28074.96843)
  MoveL 2997 to (33.29, -26.54, 130) mm, rotated rx -180 ry 0 rz 180 deg; joints [-165.409, -49.098, -91.171, 18.7, 51.788, -11.825]
  Call Extruder(28089.86428)
  MoveL 2998 to (38.36, -18.47, 130) mm, rotated rx -180 ry 0 rz 180 deg; joints [-164.468, -49.62, -89.896, 20.073, 51.279, -12.875]
  Call Extruder(28104.75993)
  MoveL 2999 to (41.5, -9.47, 130) mm, rotated rx -180 ry 0 rz 180 deg; joints [-163.355, -50.039, -88.882, 21.634, 50.982, -14.02]
  Call Extruder(28119.65580)
  MoveL 3000 to (42.57, 0, 130) mm, rotated rx 180 ry 0 rz 180 deg; joints [-162.12, -50.334, -88.173, 23.302, 50.91, -15.194]
  Call Extruder(28134.55168)
  MoveL 3001 to (41.5, 9.47, 130) mm, rotated rx -180 ry 0 rz 180 deg; joints [-160.81, -50.489, -87.802, 24.995, 51.069, -16.328]
  Call Extruder(28149.44734)
  MoveL 3002 to (38.36, 18.47, 130) mm, rotated rx 180 ry 0 rz 180 deg; joints [-159.475, -50.496, -87.784, 26.638, 51.446, -17.36]
  Call Extruder(28164.34318)
  MoveL 3003 to (33.28, 26.54, 130) mm, rotated rx 180 ry 0 rz 180 deg; joints [-158.16, -50.355, -88.121, 28.16, 52.022, -18.232]
  Call Extruder(28179.23901)
  MoveL 3004 to (26.54, 33.28, 130) mm, rotated rx 180 ry 0 rz 180 deg; joints [-156.916, -50.074, -88.797, 29.503, 52.765, -18.9]
  Call Extruder(28194.13485)
  MoveL 3005 to (18.47, 38.36, 130) mm, rotated rx -180 ry 0 rz -180 deg; joints [-155.789, -49.666, -89.783, 30.616, 53.634, -19.335]
  Call Extruder(28209.03051)
  MoveL 3006 to (9.47, 41.51, 130) mm, rotated rx 180 ry 0 rz 180 deg; joints [-154.828, -49.153, -91.034, 31.459, 54.587, -19.521]
  Call Extruder(28223.92639)
  MoveL 3007 to (0, 42.57, 130) mm, rotated rx 180 ry 0 rz 180 deg; joints [-154.081, -48.562, -92.494, 31.999, 55.574, -19.456]
  Call Extruder(28238.82226)
  MoveL 3008 to (-9.47, 41.51, 130) mm, rotated rx 180 ry 0 rz -180 deg; joints [-153.594, -47.921, -94.095, 32.21, 56.549, -19.15]
  Call Extruder(28253.71791)
  MoveL 3009 to (-18.47, 38.36, 130) mm, rotated rx 180 ry 0 rz 180 deg; joints [-153.408, -47.265, -95.763, 32.07, 57.465, -18.623]
  Call Extruder(28268.61376)
  MoveL 3010 to (-26.54, 33.28, 130) mm, rotated rx 180 ry 0 rz 180 deg; joints [-153.557, -46.625, -97.415, 31.568, 58.279, -17.903]
  Call Extruder(28283.50958)
  MoveL 3011 to (-33.29, 26.54, 130) mm, rotated rx 180 ry 0 rz 180 deg; joints [-154.059, -46.035, -98.97, 30.703, 58.954, -17.027]
  Call Extruder(28298.40543)
  MoveL 3012 to (-38.36, 18.47, 130) mm, rotated rx -180 ry 0 rz -180 deg; joints [-154.913, -45.522, -100.343, 29.492, 59.456, -16.037]
  Call Extruder(28313.30109)
  MoveL 3013 to (-41.5, 9.47, 130) mm, rotated rx -180 ry 0 rz -180 deg; joints [-156.091, -45.113, -101.458, 27.978, 59.76, -14.978]
  Call Extruder(28328.19696)
  MoveL 3014 to (-42.57, 0, 130) mm, rotated rx -180 ry 0 rz -180 deg; joints [-157.533, -44.827, -102.249, 26.228, 59.85, -13.899]
  Call Extruder(28335.75125)
  MoveL 3015 to (-42.03, -4.8, 130) mm, rotated rx 180 ry 0 rz 180 deg; joints [-158.35, -44.749, -102.467, 25.273, 59.783, -13.366]
  Set speed (130.0 mm/s)
  MoveL 3016 to (-54.1, -7.67, 130) mm, rotated rx 180 ry 0 rz 180 deg; joints [-158.024, -44.03, -104.506, 25.319, 61.05, -12.899]
  Call Extruder(28339.82387)
  Set speed (30.0 mm/s)
  MoveL 3017 to (-53.59, -12.23, 130) mm, rotated rx -180 ry 0 rz 180 deg; joints [-158.835, -43.961, -104.703, 24.384, 60.99, -12.398]
  Call Extruder(28350.75401)
  MoveL 3018 to (-49.53, -23.85, 130) mm, rotated rx 180 ry 0 rz 180 deg; joints [-161.095, -43.952, -104.73, 21.845, 60.544, -11.152]
  Call Extruder(28361.68429)
  MoveL 3019 to (-42.98, -34.27, 130) mm, rotated rx 180 ry 0 rz 180 deg; joints [-163.275, -44.127, -104.227, 19.442, 59.836, -10.058]
  Call Extruder(28372.61441)
  MoveL 3020 to (-34.27, -42.98, 130) mm, rotated rx 180 ry 0 rz 180 deg; joints [-165.21, -44.477, -103.23, 17.345, 58.899, -9.165]
  Call Extruder(28383.54469)
  MoveL 3021 to (-23.85, -49.53, 130) mm, rotated rx -180 ry 0 rz 180 deg; joints [-166.774, -44.988, -101.804, 15.69, 57.781, -8.518]
  Call Extruder(28394.47483)
  MoveL 3022 to (-12.23, -53.59, 130) mm, rotated rx 180 ry 0 rz 180 deg; joints [-167.889, -45.635, -100.039, 14.566, 56.541, -8.153]
  Call Extruder(28405.40505)
  MoveL 3023 to (0, -54.97, 130) mm, rotated rx 180 ry 0 rz 180 deg; joints [-168.526, -46.388, -98.037, 14.012, 55.24, -8.098]
  Call Extruder(28414.41206)
  MoveL 3024 to (10.08, -53.83, 130) mm, rotated rx 180 ry 0 rz 180 deg; joints [-168.668, -47.062, -96.284, 14.026, 54.173, -8.319]
  Call Extruder(28416.33527)
  MoveL 3025 to (12.23, -53.59, 130) mm, rotated rx 180 ry 0 rz 180 deg; joints [-168.697, -47.209, -95.907, 14.031, 53.945, -8.367]
  Call Extruder(28427.26541)
  MoveL 3026 to (23.85, -49.53, 130) mm, rotated rx 180 ry 0 rz 180 deg; joints [-168.436, -48.056, -93.755, 14.591, 52.721, -8.96]
  Call Extruder(28438.19569)
  MoveL 3027 to (34.27, -42.98, 130) mm, rotated rx 180 ry 0 rz 180 deg; joints [-167.797, -48.888, -91.686, 15.641, 51.631, -9.859]
  Call Extruder(28449.12581)
  MoveL 3028 to (42.98, -34.27, 130) mm, rotated rx 180 ry 0 rz 180 deg; joints [-166.837, -49.662, -89.794, 17.106, 50.731, -11.023]
  Call Extruder(28460.05609)
  MoveL 3029 to (49.53, -23.85, 130) mm, rotated rx 180 ry 0 rz 180 deg; joints [-165.618, -50.338, -88.163, 18.899, 50.071, -12.393]
  Call Extruder(28470.98623)
  MoveL 3030 to (53.59, -12.23, 130) mm, rotated rx 180 ry 0 rz -180 deg; joints [-164.2, -50.881, -86.867, 20.922, 49.685, -13.893]
  Call Extruder(28481.91645)
  MoveL 3031 to (54.97, 0, 130) mm, rotated rx -180 ry 0 rz 180 deg; joints [-162.641, -51.263, -85.962, 23.068, 49.594, -15.432]
  Call Extruder(28492.84667)
  MoveL 3032 to (53.59, 12.23, 130) mm, rotated rx 180 ry 0 rz 180 deg; joints [-160.996, -51.464, -85.487, 25.234, 49.803, -16.919]
  Call Extruder(28503.77681)
  MoveL 3033 to (49.52, 23.85, 130) mm, rotated rx 180 ry 0 rz -180 deg; joints [-159.322, -51.474, -85.464, 27.32, 50.297, -18.263]
  Call Extruder(28514.70709)
  MoveL 3034 to (42.98, 34.27, 130) mm, rotated rx 180 ry 0 rz 180 deg; joints [-157.673, -51.291, -85.895, 29.243, 51.048, -19.39]
  Call Extruder(28525.63721)
  MoveL 3035 to (34.27, 42.98, 130) mm, rotated rx -180 ry 0 rz 180 deg; joints [-156.102, -50.926, -86.759, 30.931, 52.012, -20.245]
  Call Extruder(28536.56749)
  MoveL 3036 to (23.85, 49.52, 130) mm, rotated rx -180 ry 0 rz 180 deg; joints [-154.667, -50.398, -88.019, 32.329, 53.138, -20.79]
  Call Extruder(28547.49763)
  MoveL 3037 to (12.23, 53.59, 130) mm, rotated rx 180 ry 0 rz 180 deg; joints [-153.426, -49.734, -89.619, 33.395, 54.368, -21.01]
  Call Extruder(28558.42785)
  MoveL 3038 to (0, 54.97, 130) mm, rotated rx 180 ry 0 rz 180 deg; joints [-152.438, -48.968, -91.489, 34.092, 55.639, -20.907]
  Call Extruder(28569.35808)
  MoveL 3039 to (-12.23, 53.59, 130) mm, rotated rx 180 ry 0 rz 180 deg; joints [-151.764, -48.14, -93.545, 34.389, 56.893, -20.498]
  Call Extruder(28580.28821)
  MoveL 3040 to (-23.85, 49.52, 130) mm, rotated rx -180 ry 0 rz 180 deg; joints [-151.463, -47.292, -95.692, 34.256, 58.069, -19.808]
  Call Extruder(28591.21849)
  MoveL 3041 to (-34.27, 42.98, 130) mm, rotated rx -180 ry 0 rz 180 deg; joints [-151.589, -46.467, -97.83, 33.669, 59.116, -18.877]
  Call Extruder(28602.14862)
  MoveL 3042 to (-42.98, 34.27, 130) mm, rotated rx -180 ry 0 rz -180 deg; joints [-152.179, -45.706, -99.849, 32.615, 59.984, -17.75]
  Call Extruder(28613.07889)
  MoveL 3043 to (-49.52, 23.85, 130) mm, rotated rx -180 ry 0 rz -180 deg; joints [-153.248, -45.046, -101.643, 31.098, 60.633, -16.479]
  Call Extruder(28624.00904)
  MoveL 3044 to (-53.59, 12.23, 130) mm, rotated rx 180 ry 0 rz -180 deg; joints [-154.769, -44.521, -103.106, 29.159, 61.03, -15.122]
  Call Extruder(28634.93926)
  MoveL 3045 to (-54.97, 0, 130) mm, rotated rx 180 ry 0 rz -180 deg; joints [-156.673, -44.154, -104.149, 26.878, 61.153, -13.741]
  Call Extruder(28640.46488)
  MoveL 3046 to (-54.27, -6.18, 130) mm, rotated rx 180 ry 0 rz 180 deg; joints [-157.76, -44.053, -104.439, 25.623, 61.07, -13.062]
  Set speed (130.0 mm/s)
  MoveL 3047 to (-49.9, -9.51, 130) mm, rotated rx 180 ry 0 rz -180 deg; joints [-158.616, -44.216, -103.972, 24.739, 60.604, -12.744]
  MoveL 3048 to (2.97, -12.99, 130) mm, rotated rx 180 ry 0 rz -180 deg; joints [-162.152, -47.294, -95.687, 21.963, 55.034, -13.013]
  Call Extruder(28645.12846)
  Set speed (80.0 mm/s)
  MoveL 3049 to (5.78, -12.01, 130) mm, rotated rx 180 ry 0 rz 180 deg; joints [-162.141, -47.499, -95.163, 22.06, 54.741, -13.167]
  Call Extruder(28649.79208)
  MoveL 3050 to (8.31, -10.42, 130) mm, rotated rx 180 ry 0 rz -180 deg; joints [-162.027, -47.7, -94.653, 22.279, 54.48, -13.389]
  Call Extruder(28654.45627)
  MoveL 3051 to (10.42, -8.31, 130) mm, rotated rx -180 ry 0 rz 180 deg; joints [-161.819, -47.887, -94.182, 22.606, 54.266, -13.667]
  Call Extruder(28659.11990)
  MoveL 3052 to (12.01, -5.78, 130) mm, rotated rx 180 ry 0 rz -180 deg; joints [-161.529, -48.049, -93.773, 23.022, 54.108, -13.989]
  Call Extruder(28663.78347)
  MoveL 3053 to (13, -2.97, 130) mm, rotated rx 180 ry 0 rz -180 deg; joints [-161.171, -48.179, -93.447, 23.507, 54.015, -14.336]
  Call Extruder(28668.44742)
  MoveL 3054 to (13.33, 0, 130) mm, rotated rx 180 ry 0 rz 180 deg; joints [-160.763, -48.271, -93.218, 24.035, 53.992, -14.691]
  Call Extruder(28673.11138)
  MoveL 3055 to (13, 2.97, 130) mm, rotated rx -180 ry 0 rz 180 deg; joints [-160.324, -48.319, -93.098, 24.581, 54.039, -15.036]
  Call Extruder(28677.77495)
  MoveL 3056 to (12.01, 5.78, 130) mm, rotated rx -180 ry 0 rz -180 deg; joints [-159.874, -48.321, -93.092, 25.119, 54.154, -15.352]
  Call Extruder(28682.43857)
  MoveL 3057 to (10.42, 8.31, 130) mm, rotated rx -180 ry 0 rz 180 deg; joints [-159.432, -48.278, -93.201, 25.622, 54.331, -15.624]
  Call Extruder(28687.10276)
  MoveL 3058 to (8.31, 10.42, 130) mm, rotated rx 180 ry 0 rz 180 deg; joints [-159.021, -48.19, -93.419, 26.069, 54.56, -15.837]
  Call Extruder(28691.76639)
  MoveL 3059 to (5.78, 12.01, 130) mm, rotated rx -180 ry 0 rz 180 deg; joints [-158.657, -48.064, -93.737, 26.437, 54.831, -15.981]
  Call Extruder(28696.42996)
  MoveL 3060 to (2.97, 12.99, 130) mm, rotated rx 180 ry 0 rz 180 deg; joints [-158.359, -47.904, -94.138, 26.711, 55.13, -16.05]
  Call Extruder(28701.09391)
  MoveL 3061 to (0, 13.33, 130) mm, rotated rx -180 ry 0 rz 180 deg; joints [-158.143, -47.72, -94.604, 26.877, 55.441, -16.04]
  Call Extruder(28705.75786)
  MoveL 3062 to (-2.97, 12.99, 130) mm, rotated rx -180 ry 0 rz 180 deg; joints [-158.019, -47.52, -95.112, 26.925, 55.749, -15.952]
  Call Extruder(28710.42143)
  MoveL 3063 to (-5.78, 12.01, 130) mm, rotated rx -180 ry 0 rz 180 deg; joints [-157.997, -47.314, -95.636, 26.853, 56.039, -15.793]
  Call Extruder(28715.08507)
  MoveL 3064 to (-8.31, 10.42, 130) mm, rotated rx 180 ry 0 rz 180 deg; joints [-158.08, -47.114, -96.15, 26.662, 56.297, -15.569]
  Call Extruder(28719.74926)
  MoveL 3065 to (-10.42, 8.31, 130) mm, rotated rx -180 ry 0 rz 180 deg; joints [-158.266, -46.928, -96.629, 26.36, 56.51, -15.293]
  Call Extruder(28724.41288)
  MoveL 3066 to (-12.01, 5.78, 130) mm, rotated rx 180 ry 0 rz 180 deg; joints [-158.549, -46.767, -97.047, 25.959, 56.667, -14.977]
  Call Extruder(28729.07645)
  MoveL 3067 to (-13, 2.97, 130) mm, rotated rx 180 ry 0 rz -180 deg; joints [-158.913, -46.637, -97.384, 25.478, 56.76, -14.638]
  Call Extruder(28733.74041)
  MoveL 3068 to (-13.33, 0, 130) mm, rotated rx -180 ry 0 rz 180 deg; joints [-159.341, -46.547, -97.621, 24.941, 56.785, -14.292]
  Call Extruder(28738.40436)
  MoveL 3069 to (-13, -2.97, 130) mm, rotated rx 180 ry 0 rz 180 deg; joints [-159.811, -46.499, -97.745, 24.376, 56.741, -13.956]
  Call Extruder(28743.06793)
  MoveL 3070 to (-12.01, -5.78, 130) mm, rotated rx 180 ry 0 rz 180 deg; joints [-160.294, -46.497, -97.751, 23.813, 56.629, -13.645]
  Call Extruder(28747.73156)
  MoveL 3071 to (-10.42, -8.31, 130) mm, rotated rx 180 ry 0 rz 180 deg; joints [-160.766, -46.54, -97.638, 23.282, 56.455, -13.375]
  Call Extruder(28752.39574)
  MoveL 3072 to (-8.31, -10.42, 130) mm, rotated rx 180 ry 0 rz 180 deg; joints [-161.2, -46.627, -97.412, 22.811, 56.227, -13.16]
  Call Extruder(28757.05938)
  MoveL 3073 to (-5.78, -12.01, 130) mm, rotated rx -180 ry 0 rz 180 deg; joints [-161.572, -46.752, -97.084, 22.427, 55.956, -13.01]
  Call Extruder(28761.72294)
  MoveL 3074 to (-2.97, -12.99, 130) mm, rotated rx 180 ry 0 rz 180 deg; joints [-161.863, -46.911, -96.673, 22.149, 55.657, -12.933]
  Call Extruder(28766.38690)
  MoveL 3075 to (0, -13.33, 130) mm, rotated rx -180 ry 0 rz -180 deg; joints [-162.059, -47.095, -96.199, 21.992, 55.344, -12.934]
  Call Extruder(28771.05084)
  MoveL 3076 to (2.97, -12.99, 130) mm, rotated rx 180 ry 0 rz -180 deg; joints [-162.152, -47.294, -95.687, 21.963, 55.034, -13.013]
  Set speed (130.0 mm/s)
  MoveL 3077 to (2.97, -12.99, 135) mm, rotated rx 180 ry 0 rz -180 deg; joints [-162.152, -46.543, -95.942, 22.094, 54.573, -13.241]
  MoveL 3078 to (-26.25, -4.54, 135) mm, rotated rx -180 ry 0 rz 180 deg; joints [-159.288, -44.873, -100.231, 24.749, 57.648, -13.857]
  Call Extruder(28773.28346)
  Set speed (60.0 mm/s)
  MoveL 3079 to (-26.09, -5.96, 135) mm, rotated rx -180 ry 0 rz 180 deg; joints [-159.522, -44.85, -100.29, 24.471, 57.626, -13.696]
  Call Extruder(28782.64825)
  MoveL 3080 to (-24.11, -11.61, 135) mm, rotated rx -180 ry 0 rz 180 deg; joints [-160.532, -44.846, -100.303, 23.305, 57.399, -13.066]
  Call Extruder(28792.01317)
  MoveL 3081 to (-20.93, -16.69, 135) mm, rotated rx 180 ry 0 rz 180 deg; joints [-161.513, -44.934, -100.07, 22.202, 57.049, -12.516]
  Call Extruder(28801.37838)
  MoveL 3082 to (-16.69, -20.93, 135) mm, rotated rx -180 ry 0 rz 180 deg; joints [-162.406, -45.112, -99.606, 21.229, 56.592, -12.073]
  Call Extruder(28810.74330)
  MoveL 3083 to (-11.61, -24.12, 135) mm, rotated rx 180 ry 0 rz 180 deg; joints [-163.159, -45.369, -98.936, 20.441, 56.051, -11.758]
  Call Extruder(28820.10808)
  MoveL 3084 to (-5.96, -26.09, 135) mm, rotated rx 180 ry 0 rz 180 deg; joints [-163.733, -45.694, -98.098, 19.882, 55.454, -11.589]
  Call Extruder(28829.47319)
  MoveL 3085 to (0, -26.77, 135) mm, rotated rx 180 ry 0 rz 180 deg; joints [-164.103, -46.07, -97.137, 19.578, 54.829, -11.577]
  Call Extruder(28838.83829)
  MoveL 3086 to (5.96, -26.09, 135) mm, rotated rx 180 ry 0 rz 180 deg; joints [-164.258, -46.479, -96.104, 19.54, 54.209, -11.726]
  Call Extruder(28848.20310)
  MoveL 3087 to (11.61, -24.11, 135) mm, rotated rx 180 ry 0 rz 180 deg; joints [-164.201, -46.899, -95.05, 19.765, 53.625, -12.03]
  Call Extruder(28857.56801)
  MoveL 3088 to (16.69, -20.93, 135) mm, rotated rx 180 ry 0 rz 180 deg; joints [-163.944, -47.311, -94.03, 20.233, 53.107, -12.476]
  Call Extruder(28866.93322)
  MoveL 3089 to (20.93, -16.69, 135) mm, rotated rx 180 ry 0 rz 180 deg; joints [-163.508, -47.693, -93.091, 20.914, 52.682, -13.043]
  Call Extruder(28876.29814)
  MoveL 3090 to (24.11, -11.61, 135) mm, rotated rx 180 ry 0 rz 180 deg; joints [-162.92, -48.026, -92.278, 21.769, 52.371, -13.702]
  Call Extruder(28885.66293)
  MoveL 3091 to (26.09, -5.96, 135) mm, rotated rx 180 ry 0 rz -180 deg; joints [-162.209, -48.293, -91.63, 22.751, 52.192, -14.417]
  Call Extruder(28895.02803)
  MoveL 3092 to (26.77, 0, 135) mm, rotated rx -180 ry 0 rz -180 deg; joints [-161.41, -48.481, -91.177, 23.811, 52.151, -15.15]
  Call Extruder(28904.39314)
  MoveL 3093 to (26.09, 5.96, 135) mm, rotated rx -180 ry 0 rz 180 deg; joints [-160.556, -48.579, -90.94, 24.897, 52.253, -15.861]
  Call Extruder(28913.75794)
  MoveL 3094 to (24.11, 11.61, 135) mm, rotated rx 180 ry 0 rz 180 deg; joints [-159.683, -48.584, -90.928, 25.958, 52.49, -16.511]
  Call Extruder(28923.12285)
  MoveL 3095 to (20.93, 16.69, 135) mm, rotated rx 180 ry 0 rz 180 deg; joints [-158.826, -48.494, -91.144, 26.947, 52.851, -17.066]
  Call Extruder(28932.48806)
  MoveL 3096 to (16.69, 20.93, 135) mm, rotated rx 180 ry 0 rz 180 deg; joints [-158.019, -48.315, -91.576, 27.823, 53.316, -17.499]
  Call Extruder(28941.85297)
  MoveL 3097 to (11.61, 24.11, 135) mm, rotated rx 180 ry 0 rz 180 deg; joints [-157.299, -48.056, -92.206, 28.547, 53.86, -17.788]
  Call Extruder(28951.21777)
  MoveL 3098 to (5.96, 26.09, 135) mm, rotated rx 180 ry 0 rz 180 deg; joints [-156.697, -47.729, -93.004, 29.09, 54.457, -17.922]
  Call Extruder(28960.58288)
  MoveL 3099 to (0, 26.77, 135) mm, rotated rx 180 ry 0 rz 180 deg; joints [-156.245, -47.351, -93.932, 29.427, 55.076, -17.897]
  Call Extruder(28969.94798)
